Staubli VAL3: readText.dtx

public bool bBYPASS
public bool bCycle
public bool bCycleEnd
bool bGetSpeed = true
bool bMatlab
bool bReadEnd
bool bReadWait
public bool bResumeCycle
bool bTxtHeadOk
public bool bWriteEnd
frame fPrdFrame = {fatherId=world[0]}
jointRx jJointRead[100] = {j1=8.22, j2=20.1, j3=107.19, j4=-141.77, j5=44.38, j6=150.9}
public jointRx jPrdHome
mdesc mNomSpeed = {accel=16, vel=40, decel=16, tmax=80, blend=off, leave=20, reach=20}
public mdesc mSpdOfJnt[100]
  [0] = {accel=40, vel=40, decel=40, rmax=1000, tmax=40, blend=cartesian, leave=0, reach=2}
  [1] = {accel=30, vel=40, decel=30, rmax=1000, tmax=40, blend=cartesian, leave=0, reach=2}
  [2] = {accel=30, vel=40, decel=30, rmax=1000, tmax=15.702, blend=cartesian, leave=0, reach=2}
  [3] = {accel=30, vel=40, decel=30, rmax=1000, tmax=6.112, blend=cartesian, leave=0, reach=2}
  [4] = {accel=16, vel=40, decel=16, rmax=1000, tmax=200, blend=cartesian, leave=2, reach=2}
  [5] = {accel=16, vel=40, decel=16, rmax=1000, tmax=200, blend=cartesian, leave=2, reach=2}
  [6] = {accel=16, vel=40, decel=16, rmax=1000, tmax=200, blend=cartesian, leave=2, reach=2}
  [7] = {accel=16, vel=40, decel=16, rmax=1000, tmax=200, blend=cartesian, leave=2, reach=2}
  [8] = {accel=16, vel=40, decel=16, rmax=1000, tmax=200, blend=cartesian, leave=2, reach=2}
  [9] = {accel=16, vel=40, decel=16, rmax=1000, tmax=200, blend=cartesian, leave=2, reach=2}
  [10] = {accel=16, vel=40, decel=16, rmax=1000, tmax=200, blend=cartesian, leave=2, reach=2}
  [11] = {accel=16, vel=40, decel=16, rmax=1000, tmax=200, blend=cartesian, leave=2, reach=2}
  [12] = {accel=16, vel=40, decel=16, rmax=1000, tmax=200, blend=cartesian, leave=2, reach=2}
  [13] = {accel=16, vel=40, decel=16, rmax=1000, tmax=200, blend=cartesian, leave=2, reach=2}
  [14] = {accel=16, vel=40, decel=16, rmax=1000, tmax=200, blend=cartesian, leave=2, reach=2}
  [15] = {accel=16, vel=40, decel=16, rmax=1000, tmax=200, blend=cartesian, leave=2, reach=2}
  [16] = {accel=16, vel=40, decel=16, rmax=1000, tmax=200, blend=cartesian, leave=2, reach=2}
  [17] = {accel=16, vel=40, decel=16, rmax=1000, tmax=200, blend=cartesian, leave=2, reach=2}
  [18] = {accel=16, vel=40, decel=16, rmax=1000, tmax=200, blend=cartesian, leave=2, reach=2}
  [19] = {accel=16, vel=40, decel=16, rmax=1000, tmax=200, blend=cartesian, leave=2, reach=2}
  [20] = {accel=16, vel=40, decel=16, rmax=1000, tmax=200, blend=cartesian, leave=2, reach=2}
  [21] = {accel=16, vel=40, decel=16, rmax=1000, tmax=200, blend=cartesian, leave=2, reach=2}
  [22] = {accel=16, vel=40, decel=16, rmax=1000, tmax=200, blend=cartesian, leave=2, reach=2}
  [23] = {accel=16, vel=40, decel=16, rmax=1000, tmax=200, blend=cartesian, leave=2, reach=2}
  [24] = {accel=16, vel=40, decel=16, rmax=1000, tmax=200, blend=cartesian, leave=2, reach=2}
  [25] = {accel=16, vel=40, decel=16, rmax=1000, tmax=200, blend=cartesian, leave=2, reach=2}
  [26] = {accel=16, vel=40, decel=16, rmax=1000, tmax=200, blend=cartesian, leave=2, reach=2}
  [27] = {accel=16, vel=40, decel=16, rmax=1000, tmax=200, blend=cartesian, leave=2, reach=2}
  [28] = {accel=16, vel=40, decel=16, rmax=1000, tmax=200, blend=cartesian, leave=2, reach=2}
  [29] = {accel=16, vel=40, decel=16, rmax=1000, tmax=200, blend=cartesian, leave=2, reach=2}
  [30] = {accel=16, vel=40, decel=16, rmax=1000, tmax=200, blend=cartesian, leave=2, reach=2}
  [31] = {accel=16, vel=40, decel=16, rmax=1000, tmax=200, blend=cartesian, leave=2, reach=2}
  [32] = {accel=16, vel=40, decel=16, rmax=1000, tmax=200, blend=cartesian, leave=2, reach=2}
  [33] = {accel=16, vel=40, decel=16, rmax=1000, tmax=200, blend=cartesian, leave=2, reach=2}
  [34] = {accel=16, vel=40, decel=16, rmax=1000, tmax=200, blend=cartesian, leave=2, reach=2}
  [35] = {accel=16, vel=40, decel=16, rmax=1000, tmax=200, blend=cartesian, leave=2, reach=2}
  [36] = {accel=16, vel=40, decel=16, rmax=1000, tmax=200, blend=cartesian, leave=2, reach=2}
  [37] = {accel=16, vel=40, decel=16, rmax=1000, tmax=200, blend=cartesian, leave=2, reach=2}
  [38] = {accel=16, vel=40, decel=16, rmax=1000, tmax=200, blend=cartesian, leave=2, reach=2}
  [39] = {accel=16, vel=40, decel=16, rmax=1000, tmax=200, blend=cartesian, leave=2, reach=2}
  [40] = {accel=16, vel=40, decel=16, rmax=1000, tmax=200, blend=cartesian, leave=2, reach=2}
  [41] = {accel=16, vel=40, decel=16, rmax=1000, tmax=200, blend=cartesian, leave=2, reach=2}
  [42] = {accel=16, vel=40, decel=16, rmax=1000, tmax=200, blend=cartesian, leave=2, reach=2}
  [43] = {accel=16, vel=40, decel=16, rmax=1000, tmax=200, blend=cartesian, leave=2, reach=2}
  [44] = {accel=16, vel=40, decel=16, rmax=1000, tmax=200, blend=cartesian, leave=2, reach=2}
  [45] = {accel=16, vel=40, decel=16, rmax=1000, tmax=200, blend=cartesian, leave=2, reach=2}
  [46] = {accel=16, vel=40, decel=16, rmax=1000, tmax=200, blend=cartesian, leave=2, reach=2}
  [47] = {accel=16, vel=40, decel=16, rmax=1000, tmax=200, blend=cartesian, leave=2, reach=2}
  [48] = {accel=16, vel=40, decel=16, rmax=1000, tmax=200, blend=cartesian, leave=2, reach=2}
  [49] = {accel=16, vel=40, decel=16, rmax=1000, tmax=200, blend=cartesian, leave=2, reach=2}
  [50] = {accel=16, vel=40, decel=16, rmax=1000, tmax=200, blend=cartesian, leave=2, reach=2}
  [51] = {accel=16, vel=40, decel=16, rmax=1000, tmax=200, blend=cartesian, leave=2, reach=2}
  [52] = {accel=16, vel=40, decel=16, rmax=1000, tmax=200, blend=cartesian, leave=2, reach=2}
  [53] = {accel=16, vel=40, decel=16, rmax=1000, tmax=200, blend=cartesian, leave=2, reach=2}
  [54] = {accel=16, vel=40, decel=16, rmax=1000, tmax=200, blend=cartesian, leave=2, reach=2}
  [55] = {accel=16, vel=40, decel=16, rmax=1000, tmax=200, blend=cartesian, leave=2, reach=2}
  [56] = {accel=16, vel=40, decel=16, rmax=1000, tmax=200, blend=cartesian, leave=2, reach=2}
  [57] = {accel=16, vel=40, decel=16, rmax=1000, tmax=200, blend=cartesian, leave=2, reach=2}
  [58] = {accel=16, vel=40, decel=16, rmax=1000, tmax=200, blend=cartesian, leave=2, reach=2}
  [59] = {accel=16, vel=40, decel=16, rmax=1000, tmax=200, blend=cartesian, leave=2, reach=2}
  [60] = {accel=16, vel=40, decel=16, rmax=1000, tmax=200, blend=cartesian, leave=2, reach=2}
  [61] = {accel=16, vel=40, decel=16, rmax=1000, tmax=200, blend=cartesian, leave=2, reach=2}
  [62] = {accel=16, vel=40, decel=16, rmax=1000, tmax=200, blend=cartesian, leave=2, reach=2}
  [63] = {accel=16, vel=40, decel=16, rmax=1000, tmax=200, blend=cartesian, leave=2, reach=2}
  [64] = {accel=16, vel=40, decel=16, rmax=1000, tmax=200, blend=cartesian, leave=2, reach=2}
  [65] = {accel=16, vel=40, decel=16, rmax=1000, tmax=200, blend=cartesian, leave=2, reach=2}
  [66] = {accel=16, vel=40, decel=16, rmax=1000, tmax=200, blend=cartesian, leave=2, reach=2}
  [67] = {accel=16, vel=40, decel=16, rmax=1000, tmax=200, blend=cartesian, leave=2, reach=2}
  [68] = {accel=16, vel=40, decel=16, rmax=1000, tmax=200, blend=cartesian, leave=2, reach=2}
  [69] = {accel=16, vel=40, decel=16, rmax=1000, tmax=200, blend=cartesian, leave=2, reach=2}
  [70] = {accel=16, vel=40, decel=16, rmax=1000, tmax=200, blend=cartesian, leave=2, reach=2}
  [71] = {accel=16, vel=40, decel=16, rmax=1000, tmax=200, blend=cartesian, leave=2, reach=2}
  [72] = {accel=16, vel=40, decel=16, rmax=1000, tmax=200, blend=cartesian, leave=2, reach=2}
  [73] = {accel=16, vel=40, decel=16, rmax=1000, tmax=200, blend=cartesian, leave=2, reach=2}
  [74] = {accel=16, vel=40, decel=16, rmax=1000, tmax=200, blend=cartesian, leave=2, reach=2}
  [75] = {accel=16, vel=40, decel=16, rmax=1000, tmax=200, blend=cartesian, leave=2, reach=2}
  [76] = {accel=16, vel=40, decel=16, rmax=1000, tmax=200, blend=cartesian, leave=2, reach=2}
  [77] = {accel=16, vel=40, decel=16, rmax=1000, tmax=200, blend=cartesian, leave=2, reach=2}
  [78] = {accel=16, vel=40, decel=16, rmax=1000, tmax=200, blend=cartesian, leave=2, reach=2}
  [79] = {accel=16, vel=40, decel=16, rmax=1000, tmax=200, blend=cartesian, leave=2, reach=2}
  [80] = {accel=16, vel=40, decel=16, rmax=1000, tmax=200, blend=cartesian, leave=2, reach=2}
  [81] = {accel=16, vel=40, decel=16, rmax=1000, tmax=200, blend=cartesian, leave=2, reach=2}
  [82] = {accel=16, vel=40, decel=16, rmax=1000, tmax=200, blend=cartesian, leave=2, reach=2}
  [83] = {accel=16, vel=40, decel=16, rmax=1000, tmax=200, blend=cartesian, leave=2, reach=2}
  [84] = {accel=16, vel=40, decel=16, rmax=1000, tmax=200, blend=cartesian, leave=2, reach=2}
  [85] = {accel=16, vel=40, decel=16, rmax=1000, tmax=200, blend=cartesian, leave=2, reach=2}
  [86] = {accel=16, vel=40, decel=16, rmax=1000, tmax=200, blend=cartesian, leave=2, reach=2}
  [87] = {accel=16, vel=40, decel=16, rmax=1000, tmax=200, blend=cartesian, leave=2, reach=2}
  [88] = {accel=16, vel=40, decel=16, rmax=1000, tmax=200, blend=cartesian, leave=2, reach=2}
  [89] = {accel=16, vel=40, decel=16, rmax=1000, tmax=200, blend=cartesian, leave=2, reach=2}
  [90] = {accel=16, vel=40, decel=16, rmax=1000, tmax=200, blend=cartesian, leave=2, reach=2}
  [91] = {accel=16, vel=40, decel=16, rmax=1000, tmax=200, blend=cartesian, leave=2, reach=2}
  [92] = {accel=16, vel=40, decel=16, rmax=1000, tmax=200, blend=cartesian, leave=2, reach=2}
  [93] = {accel=16, vel=40, decel=16, rmax=1000, tmax=200, blend=cartesian, leave=2, reach=2}
  [94] = {accel=16, vel=40, decel=16, rmax=1000, tmax=200, blend=cartesian, leave=2, reach=2}
  [95] = {accel=16, vel=40, decel=16, rmax=1000, tmax=200, blend=cartesian, leave=2, reach=2}
  [96] = {accel=16, vel=40, decel=16, rmax=1000, tmax=200, blend=cartesian, leave=2, reach=2}
  [97] = {accel=16, vel=40, decel=16, rmax=1000, tmax=200, blend=cartesian, leave=2, reach=2}
  [98] = {accel=16, vel=40, decel=16, rmax=1000, tmax=200, blend=cartesian, leave=2, reach=2}
  [99] = {accel=16, vel=40, decel=16, rmax=1000, tmax=200, blend=cartesian, leave=2, reach=2}
public mdesc mSpdOfPt[1000]
  [0] = {accel=30, decel=30, tmax=100, leave=0, reach=0.5}
  [1] = {accel=80, decel=80, tmax=40, leave=0.5, reach=0.5}
  [2] = {accel=80, decel=80, tmax=20, leave=2, reach=0.5}
  [3] = {accel=80, decel=80, tmax=6.283, leave=0, reach=0.5}
  [4] = {accel=80, decel=80, tmax=9.415, leave=0, reach=0.5}
  [5] = {accel=80, decel=80, tmax=9.426, leave=0, reach=0.5}
  [6] = {accel=80, decel=80, tmax=9.491, leave=0, reach=0.5}
  [7] = {accel=80, decel=80, tmax=9.63, leave=0, reach=0.5}
  [8] = {accel=80, decel=80, tmax=9.837, leave=0, reach=0.5}
  [9] = {accel=80, decel=80, tmax=10.085, leave=0, reach=0.5}
  [10] = {accel=80, decel=80, tmax=10.343, leave=0, reach=0.5}
  [11] = {accel=80, decel=80, tmax=10.597, leave=0, reach=0.5}
  [12] = {accel=80, decel=80, tmax=10.851, leave=0, reach=0.5}
  [13] = {accel=80, decel=80, tmax=11.121, leave=0, reach=0.5}
  [14] = {accel=80, decel=80, tmax=11.43, leave=0, reach=0.5}
  [15] = {accel=80, decel=80, tmax=11.774, leave=0, reach=0.5}
  [16] = {accel=80, decel=80, tmax=12.135, leave=0, reach=0.5}
  [17] = {accel=80, decel=80, tmax=12.558, leave=0, reach=0.5}
  [18] = {accel=80, decel=80, tmax=13.049, leave=0, reach=0.5}
  [19] = {accel=80, decel=80, tmax=13.543, leave=0, reach=0.5}
  [20] = {accel=80, decel=80, tmax=14.016, leave=0, reach=0.5}
  [21] = {accel=80, decel=80, tmax=14.458, leave=0, reach=0.5}
  [22] = {accel=80, decel=80, tmax=14.885, leave=0, reach=0.5}
  [23] = {accel=80, decel=80, tmax=15.328, leave=0, reach=0.5}
  [24] = {accel=80, decel=80, tmax=15.823, leave=0, reach=0.5}
  [25] = {accel=80, decel=80, tmax=16.391, leave=0, reach=0.5}
  [26] = {accel=80, decel=80, tmax=17.025, leave=0, reach=0.5}
  [27] = {accel=80, decel=80, tmax=17.694, leave=0, reach=0.5}
  [28] = {accel=80, decel=80, tmax=80, leave=0, reach=0.5}
  [29] = {accel=80, decel=80, tmax=22.598, leave=0, reach=0.5}
  [30] = {accel=80, decel=80, tmax=22.402, leave=0, reach=0.5}
  [31] = {accel=80, decel=80, tmax=21.992, leave=0, reach=0.5}
  [32] = {accel=80, decel=80, tmax=21.406, leave=0, reach=0.5}
  [33] = {accel=80, decel=80, tmax=20.689, leave=0, reach=0.5}
  [34] = {accel=80, decel=80, tmax=19.887, leave=0, reach=0.5}
  [35] = {accel=80, decel=80, tmax=19.047, leave=0, reach=0.5}
  [36] = {accel=80, decel=80, tmax=18.222, leave=0, reach=0.5}
  [37] = {accel=80, decel=80, tmax=17.459, leave=0, reach=0.5}
  [38] = {accel=80, decel=80, tmax=16.784, leave=0, reach=0.5}
  [39] = {accel=80, decel=80, tmax=16.194, leave=0, reach=0.5}
  [40] = {accel=80, decel=80, tmax=15.663, leave=0, reach=0.5}
  [41] = {accel=80, decel=80, tmax=15.153, leave=0, reach=0.5}
  [42] = {accel=80, decel=80, tmax=14.634, leave=0, reach=0.5}
  [43] = {accel=80, decel=80, tmax=14.096, leave=0, reach=0.5}
  [44] = {accel=80, decel=80, tmax=13.551, leave=0, reach=0.5}
  [45] = {accel=80, decel=80, tmax=13.023, leave=0, reach=0.5}
  [46] = {accel=80, decel=80, tmax=12.575, leave=0, reach=0.5}
  [47] = {accel=80, decel=80, tmax=12.194, leave=0, reach=0.5}
  [48] = {accel=80, decel=80, tmax=11.83, leave=0, reach=0.5}
  [49] = {accel=80, decel=80, tmax=11.503, leave=0, reach=0.5}
  [50] = {accel=80, decel=80, tmax=11.215, leave=0, reach=0.5}
  [51] = {accel=80, decel=80, tmax=10.948, leave=0, reach=0.5}
  [52] = {accel=80, decel=80, tmax=10.683, leave=0, reach=0.5}
  [53] = {accel=80, decel=80, tmax=10.416, leave=0, reach=0.5}
  [54] = {accel=80, decel=80, tmax=10.16, leave=0, reach=0.5}
  [55] = {accel=80, decel=80, tmax=9.943, leave=0, reach=0.5}
  [56] = {accel=80, decel=80, tmax=9.794, leave=0, reach=0.5}
  [57] = {accel=80, decel=80, tmax=9.721, leave=0, reach=0.5}
  [58] = {accel=80, decel=80, tmax=9.707, leave=0, reach=0.5}
  [59] = {accel=80, decel=80, tmax=9.72, leave=0, reach=0.5}
  [60] = {accel=80, decel=80, tmax=9.72, leave=0, reach=0.5}
  [61] = {accel=80, decel=80, tmax=9.688, leave=0, reach=0.5}
  [62] = {accel=80, decel=80, tmax=9.617, leave=0, reach=0.5}
  [63] = {accel=80, decel=80, tmax=9.515, leave=0, reach=0.5}
  [64] = {accel=80, decel=80, tmax=9.389, leave=0, reach=0.5}
  [65] = {accel=80, decel=80, tmax=46.527, leave=0, reach=0.5}
  [66] = {accel=80, decel=80, tmax=8.998, leave=0, reach=0.5}
  [67] = {accel=80, decel=80, tmax=9.118, leave=0, reach=0.5}
  [68] = {accel=80, decel=80, tmax=9.246, leave=0, reach=0.5}
  [69] = {accel=80, decel=80, tmax=9.386, leave=0, reach=0.5}
  [70] = {accel=80, decel=80, tmax=9.534, leave=0, reach=0.5}
  [71] = {accel=80, decel=80, tmax=9.678, leave=0, reach=0.5}
  [72] = {accel=80, decel=80, tmax=9.805, leave=0, reach=0.5}
  [73] = {accel=80, decel=80, tmax=9.903, leave=0, reach=0.5}
  [74] = {accel=80, decel=80, tmax=9.967, leave=0, reach=0.5}
  [75] = {accel=80, decel=80, tmax=9.994, leave=0, reach=0.5}
  [76] = {accel=80, decel=80, tmax=9.995, leave=0, reach=0.5}
  [77] = {accel=80, decel=80, tmax=9.992, leave=0, reach=0.5}
  [78] = {accel=80, decel=80, tmax=10.02, leave=0, reach=0.5}
  [79] = {accel=80, decel=80, tmax=10.106, leave=0, reach=0.5}
  [80] = {accel=80, decel=80, tmax=10.26, leave=0, reach=0.5}
  [81] = {accel=80, decel=80, tmax=10.472, leave=0, reach=0.5}
  [82] = {accel=80, decel=80, tmax=10.718, leave=0, reach=0.5}
  [83] = {accel=80, decel=80, tmax=10.977, leave=0, reach=0.5}
  [84] = {accel=80, decel=80, tmax=11.242, leave=0, reach=0.5}
  [85] = {accel=80, decel=80, tmax=11.521, leave=0, reach=0.5}
  [86] = {accel=80, decel=80, tmax=11.83, leave=0, reach=0.5}
  [87] = {accel=80, decel=80, tmax=12.182, leave=0, reach=0.5}
  [88] = {accel=80, decel=80, tmax=12.568, leave=0, reach=0.5}
  [89] = {accel=80, decel=80, tmax=12.965, leave=0, reach=0.5}
  [90] = {accel=80, decel=80, tmax=13.429, leave=0, reach=0.5}
  [91] = {accel=80, decel=80, tmax=13.979, leave=0, reach=0.5}
  [92] = {accel=80, decel=80, tmax=14.561, leave=0, reach=0.5}
  [93] = {accel=80, decel=80, tmax=15.156, leave=0, reach=0.5}
  [94] = {accel=80, decel=80, tmax=15.752, leave=0, reach=0.5}
  [95] = {accel=80, decel=80, tmax=16.352, leave=0, reach=0.5}
  [96] = {accel=80, decel=80, tmax=16.979, leave=0, reach=0.5}
  [97] = {accel=80, decel=80, tmax=17.664, leave=0, reach=0.5}
  [98] = {accel=80, decel=80, tmax=18.437, leave=0, reach=0.5}
  [99] = {accel=80, decel=80, tmax=19.31, leave=0, reach=0.5}
  [100] = {accel=80, decel=80, tmax=20.273, leave=0, reach=0.5}
  [101] = {accel=80, decel=80, tmax=21.286, leave=0, reach=0.5}
  [102] = {accel=80, decel=80, tmax=22.298, leave=0, reach=0.5}
  [103] = {accel=80, decel=80, tmax=23.255, leave=0, reach=0.5}
  [104] = {accel=80, decel=80, tmax=24.103, leave=0, reach=0.5}
  [105] = {accel=80, decel=80, tmax=24.781, leave=0, reach=0.5}
  [106] = {accel=80, decel=80, tmax=25.228, leave=0, reach=0.5}
  [107] = {accel=80, decel=80, tmax=25.404, leave=0, reach=0.5}
  [108] = {accel=80, decel=80, tmax=25.299, leave=0, reach=0.5}
  [109] = {accel=80, decel=80, tmax=24.922, leave=0, reach=0.5}
  [110] = {accel=80, decel=80, tmax=24.286, leave=0, reach=0.5}
  [111] = {accel=80, decel=80, tmax=75.027, leave=0, reach=0.5}
  [112] = {accel=80, decel=80, tmax=24.232, leave=0, reach=0.5}
  [113] = {accel=80, decel=80, tmax=25.564, leave=0, reach=0.5}
  [114] = {accel=80, decel=80, tmax=26.713, leave=0, reach=0.5}
  [115] = {accel=80, decel=80, tmax=27.589, leave=0, reach=0.5}
  [116] = {accel=80, decel=80, tmax=28.14, leave=0, reach=0.5}
  [117] = {accel=80, decel=80, tmax=28.354, leave=0, reach=0.5}
  [118] = {accel=80, decel=80, tmax=28.23, leave=0, reach=0.5}
  [119] = {accel=80, decel=80, tmax=27.776, leave=0, reach=0.5}
  [120] = {accel=80, decel=80, tmax=27.029, leave=0, reach=0.5}
  [121] = {accel=80, decel=80, tmax=26.056, leave=0, reach=0.5}
  [122] = {accel=80, decel=80, tmax=24.937, leave=0, reach=0.5}
  [123] = {accel=80, decel=80, tmax=23.743, leave=0, reach=0.5}
  [124] = {accel=80, decel=80, tmax=22.534, leave=0, reach=0.5}
  [125] = {accel=80, decel=80, tmax=21.368, leave=0, reach=0.5}
  [126] = {accel=80, decel=80, tmax=20.288, leave=0, reach=0.5}
  [127] = {accel=80, decel=80, tmax=19.318, leave=0, reach=0.5}
  [128] = {accel=80, decel=80, tmax=18.454, leave=0, reach=0.5}
  [129] = {accel=80, decel=80, tmax=17.673, leave=0, reach=0.5}
  [130] = {accel=80, decel=80, tmax=16.951, leave=0, reach=0.5}
  [131] = {accel=80, decel=80, tmax=16.265, leave=0, reach=0.5}
  [132] = {accel=80, decel=80, tmax=15.601, leave=0, reach=0.5}
  [133] = {accel=80, decel=80, tmax=14.96, leave=0, reach=0.5}
  [134] = {accel=80, decel=80, tmax=14.352, leave=0, reach=0.5}
  [135] = {accel=80, decel=80, tmax=13.787, leave=0, reach=0.5}
  [136] = {accel=80, decel=80, tmax=13.313, leave=0, reach=0.5}
  [137] = {accel=80, decel=80, tmax=12.9, leave=0, reach=0.5}
  [138] = {accel=80, decel=80, tmax=12.491, leave=0, reach=0.5}
  [139] = {accel=80, decel=80, tmax=12.111, leave=0, reach=0.5}
  [140] = {accel=80, decel=80, tmax=11.779, leave=0, reach=0.5}
  [141] = {accel=80, decel=80, tmax=11.485, leave=0, reach=0.5}
  [142] = {accel=80, decel=80, tmax=11.218, leave=0, reach=0.5}
  [143] = {accel=80, decel=80, tmax=10.971, leave=0, reach=0.5}
  [144] = {accel=80, decel=80, tmax=10.743, leave=0, reach=0.5}
  [145] = {accel=80, decel=80, tmax=10.546, leave=0, reach=0.5}
  [146] = {accel=80, decel=80, tmax=10.395, leave=0, reach=0.5}
  [147] = {accel=80, decel=80, tmax=10.3, leave=0, reach=0.5}
  [148] = {accel=80, decel=80, tmax=10.256, leave=0, reach=0.5}
  [149] = {accel=80, decel=80, tmax=10.244, leave=0, reach=0.5}
  [150] = {accel=80, decel=80, tmax=10.237, leave=0, reach=0.5}
  [151] = {accel=80, decel=80, tmax=10.212, leave=0, reach=0.5}
  [152] = {accel=80, decel=80, tmax=10.153, leave=0, reach=0.5}
  [153] = {accel=80, decel=80, tmax=10.056, leave=0, reach=0.5}
  [154] = {accel=80, decel=80, tmax=9.924, leave=0, reach=0.5}
  [155] = {accel=80, decel=80, tmax=9.77, leave=0, reach=0.5}
  [156] = {accel=80, decel=80, tmax=9.616, leave=0, reach=0.5}
  [157] = {accel=80, decel=80, tmax=9.484, leave=0, reach=0.5}
  [158] = {accel=80, decel=80, tmax=9.383, leave=0, reach=0.5}
  [159] = {accel=80, decel=80, tmax=9.304, leave=0, reach=0.5}
  [160] = {accel=80, decel=80, tmax=9.229, leave=0, reach=0.5}
  [161] = {accel=80, decel=80, tmax=9.137, leave=0, reach=0.5}
  [162] = {accel=80, decel=80, tmax=9.012, leave=0, reach=0.5}
  [163] = {accel=80, decel=80, tmax=28.213, leave=0, reach=0.5}
  [164] = {accel=80, decel=80, tmax=8.988, leave=0, reach=0.5}
  [165] = {accel=80, decel=80, tmax=9.149, leave=0, reach=0.5}
  [166] = {accel=80, decel=80, tmax=9.308, leave=0, reach=0.5}
  [167] = {accel=80, decel=80, tmax=9.436, leave=0, reach=0.5}
  [168] = {accel=80, decel=80, tmax=9.518, leave=0, reach=0.5}
  [169] = {accel=80, decel=80, tmax=9.559, leave=0, reach=0.5}
  [170] = {accel=80, decel=80, tmax=9.58, leave=0, reach=0.5}
  [171] = {accel=80, decel=80, tmax=9.614, leave=0, reach=0.5}
  [172] = {accel=80, decel=80, tmax=9.691, leave=0, reach=0.5}
  [173] = {accel=80, decel=80, tmax=9.819, leave=0, reach=0.5}
  [174] = {accel=80, decel=80, tmax=9.982, leave=0, reach=0.5}
  [175] = {accel=80, decel=80, tmax=10.147, leave=0, reach=0.5}
  [176] = {accel=80, decel=80, tmax=10.285, leave=0, reach=0.5}
  [177] = {accel=80, decel=80, tmax=10.38, leave=0, reach=0.5}
  [178] = {accel=80, decel=80, tmax=10.433, leave=0, reach=0.5}
  [179] = {accel=80, decel=80, tmax=10.454, leave=0, reach=0.5}
  [180] = {accel=80, decel=80, tmax=10.462, leave=0, reach=0.5}
  [181] = {accel=80, decel=80, tmax=10.479, leave=0, reach=0.5}
  [182] = {accel=80, decel=80, tmax=10.528, leave=0, reach=0.5}
  [183] = {accel=80, decel=80, tmax=10.621, leave=0, reach=0.5}
  [184] = {accel=80, decel=80, tmax=10.76, leave=0, reach=0.5}
  [185] = {accel=80, decel=80, tmax=10.941, leave=0, reach=0.5}
  [186] = {accel=80, decel=80, tmax=11.155, leave=0, reach=0.5}
  [187] = {accel=80, decel=80, tmax=11.399, leave=0, reach=0.5}
  [188] = {accel=80, decel=80, tmax=11.674, leave=0, reach=0.5}
  [189] = {accel=80, decel=80, tmax=11.989, leave=0, reach=0.5}
  [190] = {accel=80, decel=80, tmax=12.349, leave=0, reach=0.5}
  [191] = {accel=80, decel=80, tmax=12.758, leave=0, reach=0.5}
  [192] = {accel=80, decel=80, tmax=13.191, leave=0, reach=0.5}
  [193] = {accel=80, decel=80, tmax=13.618, leave=0, reach=0.5}
  [194] = {accel=80, decel=80, tmax=14.103, leave=0, reach=0.5}
  [195] = {accel=80, decel=80, tmax=14.68, leave=0, reach=0.5}
  [196] = {accel=80, decel=80, tmax=15.307, leave=0, reach=0.5}
  [197] = {accel=80, decel=80, tmax=15.981, leave=0, reach=0.5}
  [198] = {accel=80, decel=80, tmax=16.697, leave=0, reach=0.5}
  [199] = {accel=80, decel=80, tmax=17.456, leave=0, reach=0.5}
  [200] = {accel=80, decel=80, tmax=18.265, leave=0, reach=0.5}
  [201] = {accel=80, decel=80, tmax=19.14, leave=0, reach=0.5}
  [202] = {accel=80, decel=80, tmax=20.1, leave=0, reach=0.5}
  [203] = {accel=80, decel=80, tmax=21.165, leave=0, reach=0.5}
  [204] = {accel=80, decel=80, tmax=22.354, leave=0, reach=0.5}
  [205] = {accel=80, decel=80, tmax=23.661, leave=0, reach=0.5}
  [206] = {accel=80, decel=80, tmax=25.052, leave=0, reach=0.5}
  [207] = {accel=80, decel=80, tmax=26.473, leave=0, reach=0.5}
  [208] = {accel=80, decel=80, tmax=27.858, leave=0, reach=0.5}
  [209] = {accel=80, decel=80, tmax=29.13, leave=0, reach=0.5}
  [210] = {accel=80, decel=80, tmax=30.198, leave=0, reach=0.5}
  [211] = {accel=80, decel=80, tmax=30.973, leave=0, reach=0.5}
  [212] = {accel=80, decel=80, tmax=31.392, leave=0, reach=0.5}
  [213] = {accel=80, decel=80, tmax=31.427, leave=0, reach=0.5}
  [214] = {accel=80, decel=80, tmax=31.052, leave=0, reach=0.5}
  [215] = {accel=80, decel=80, tmax=30.253, leave=0, reach=0.5}
  [216] = {accel=80, decel=80, tmax=29.062, leave=0, reach=0.5}
  [217] = {accel=80, decel=80, tmax=27.585, leave=0, reach=0.5}
  [218] = {accel=80, decel=80, tmax=25.953, leave=0, reach=0.5}
  [219] = {accel=80, decel=80, tmax=24.265, leave=0, reach=0.5}
  [220] = {accel=80, decel=80, tmax=22.574, leave=0, reach=0.5}
  [221] = {accel=80, decel=80, tmax=63.913, leave=0, reach=0.5}
  [222] = {accel=80, decel=80, tmax=19.723, leave=0, reach=0.5}
  [223] = {accel=80, decel=80, tmax=21.535, leave=0, reach=0.5}
  [224] = {accel=80, decel=80, tmax=23.435, leave=0, reach=0.5}
  [225] = {accel=80, decel=80, tmax=25.393, leave=0, reach=0.5}
  [226] = {accel=80, decel=80, tmax=27.381, leave=0, reach=0.5}
  [227] = {accel=80, decel=80, tmax=29.346, leave=0, reach=0.5}
  [228] = {accel=80, decel=80, tmax=31.196, leave=0, reach=0.5}
  [229] = {accel=80, decel=80, tmax=32.785, leave=0, reach=0.5}
  [230] = {accel=80, decel=80, tmax=33.949, leave=0, reach=0.5}
  [231] = {accel=80, decel=80, tmax=34.591, leave=0, reach=0.5}
  [232] = {accel=80, decel=80, tmax=34.718, leave=0, reach=0.5}
  [233] = {accel=80, decel=80, tmax=34.385, leave=0, reach=0.5}
  [234] = {accel=80, decel=80, tmax=33.637, leave=0, reach=0.5}
  [235] = {accel=80, decel=80, tmax=32.521, leave=0, reach=0.5}
  [236] = {accel=80, decel=80, tmax=31.12, leave=0, reach=0.5}
  [237] = {accel=80, decel=80, tmax=29.544, leave=0, reach=0.5}
  [238] = {accel=80, decel=80, tmax=27.893, leave=0, reach=0.5}
  [239] = {accel=80, decel=80, tmax=26.25, leave=0, reach=0.5}
  [240] = {accel=80, decel=80, tmax=24.68, leave=0, reach=0.5}
  [241] = {accel=80, decel=80, tmax=23.233, leave=0, reach=0.5}
  [242] = {accel=80, decel=80, tmax=21.927, leave=0, reach=0.5}
  [243] = {accel=80, decel=80, tmax=20.755, leave=0, reach=0.5}
  [244] = {accel=80, decel=80, tmax=19.695, leave=0, reach=0.5}
  [245] = {accel=80, decel=80, tmax=18.727, leave=0, reach=0.5}
  [246] = {accel=80, decel=80, tmax=17.841, leave=0, reach=0.5}
  [247] = {accel=80, decel=80, tmax=17.027, leave=0, reach=0.5}
  [248] = {accel=80, decel=80, tmax=16.274, leave=0, reach=0.5}
  [249] = {accel=80, decel=80, tmax=15.579, leave=0, reach=0.5}
  [250] = {accel=80, decel=80, tmax=14.94, leave=0, reach=0.5}
  [251] = {accel=80, decel=80, tmax=14.354, leave=0, reach=0.5}
  [252] = {accel=80, decel=80, tmax=13.859, leave=0, reach=0.5}
  [253] = {accel=80, decel=80, tmax=13.416, leave=0, reach=0.5}
  [254] = {accel=80, decel=80, tmax=12.961, leave=0, reach=0.5}
  [255] = {accel=80, decel=80, tmax=12.525, leave=0, reach=0.5}
  [256] = {accel=80, decel=80, tmax=12.137, leave=0, reach=0.5}
  [257] = {accel=80, decel=80, tmax=11.798, leave=0, reach=0.5}
  [258] = {accel=80, decel=80, tmax=11.507, leave=0, reach=0.5}
  [259] = {accel=80, decel=80, tmax=11.259, leave=0, reach=0.5}
  [260] = {accel=80, decel=80, tmax=11.051, leave=0, reach=0.5}
  [261] = {accel=80, decel=80, tmax=10.884, leave=0, reach=0.5}
  [262] = {accel=80, decel=80, tmax=10.761, leave=0, reach=0.5}
  [263] = {accel=80, decel=80, tmax=10.683, leave=0, reach=0.5}
  [264] = {accel=80, decel=80, tmax=10.647, leave=0, reach=0.5}
  [265] = {accel=80, decel=80, tmax=10.64, leave=0, reach=0.5}
  [266] = {accel=80, decel=80, tmax=10.643, leave=0, reach=0.5}
  [267] = {accel=80, decel=80, tmax=10.634, leave=0, reach=0.5}
  [268] = {accel=80, decel=80, tmax=10.593, leave=0, reach=0.5}
  [269] = {accel=80, decel=80, tmax=10.507, leave=0, reach=0.5}
  [270] = {accel=80, decel=80, tmax=10.374, leave=0, reach=0.5}
  [271] = {accel=80, decel=80, tmax=10.205, leave=0, reach=0.5}
  [272] = {accel=80, decel=80, tmax=10.035, leave=0, reach=0.5}
  [273] = {accel=80, decel=80, tmax=9.904, leave=0, reach=0.5}
  [274] = {accel=80, decel=80, tmax=9.84, leave=0, reach=0.5}
  [275] = {accel=80, decel=80, tmax=9.839, leave=0, reach=0.5}
  [276] = {accel=80, decel=80, tmax=9.866, leave=0, reach=0.5}
  [277] = {accel=80, decel=80, tmax=9.877, leave=0, reach=0.5}
  [278] = {accel=80, decel=80, tmax=9.841, leave=0, reach=0.5}
  [279] = {accel=80, decel=80, tmax=9.75, leave=0, reach=0.5}
  [280] = {accel=80, decel=80, tmax=9.622, leave=0, reach=0.5}
  [281] = {accel=80, decel=80, tmax=9.483, leave=0, reach=0.5}
  [282] = {accel=80, decel=80, tmax=9.36, leave=0, reach=0.5}
  [283] = {accel=80, decel=80, tmax=9.27, leave=0, reach=0.5}
  [284] = {accel=80, decel=80, tmax=9.213, leave=0, reach=0.5}
  [285] = {accel=80, decel=80, tmax=21.042, leave=0, reach=0.5}
  [286] = {accel=80, decel=80, tmax=9.663, leave=0, reach=0.5}
  [287] = {accel=80, decel=80, tmax=9.685, leave=0, reach=0.5}
  [288] = {accel=80, decel=80, tmax=9.712, leave=0, reach=0.5}
  [289] = {accel=80, decel=80, tmax=9.76, leave=0, reach=0.5}
  [290] = {accel=80, decel=80, tmax=9.837, leave=0, reach=0.5}
  [291] = {accel=80, decel=80, tmax=9.942, leave=0, reach=0.5}
  [292] = {accel=80, decel=80, tmax=10.057, leave=0, reach=0.5}
  [293] = {accel=80, decel=80, tmax=10.157, leave=0, reach=0.5}
  [294] = {accel=80, decel=80, tmax=10.214, leave=0, reach=0.5}
  [295] = {accel=80, decel=80, tmax=10.212, leave=0, reach=0.5}
  [296] = {accel=80, decel=80, tmax=10.163, leave=0, reach=0.5}
  [297] = {accel=80, decel=80, tmax=10.107, leave=0, reach=0.5}
  [298] = {accel=80, decel=80, tmax=10.096, leave=0, reach=0.5}
  [299] = {accel=80, decel=80, tmax=10.159, leave=0, reach=0.5}
  [300] = {accel=80, decel=80, tmax=10.292, leave=0, reach=0.5}
  [301] = {accel=80, decel=80, tmax=10.456, leave=0, reach=0.5}
  [302] = {accel=80, decel=80, tmax=10.607, leave=0, reach=0.5}
  [303] = {accel=80, decel=80, tmax=10.718, leave=0, reach=0.5}
  [304] = {accel=80, decel=80, tmax=10.78, leave=0, reach=0.5}
  [305] = {accel=80, decel=80, tmax=10.8, leave=0, reach=0.5}
  [306] = {accel=80, decel=80, tmax=10.789, leave=0, reach=0.5}
  [307] = {accel=80, decel=80, tmax=10.764, leave=0, reach=0.5}
  [308] = {accel=80, decel=80, tmax=10.748, leave=0, reach=0.5}
  [309] = {accel=80, decel=80, tmax=10.761, leave=0, reach=0.5}
  [310] = {accel=80, decel=80, tmax=10.815, leave=0, reach=0.5}
  [311] = {accel=80, decel=80, tmax=10.918, leave=0, reach=0.5}
  [312] = {accel=80, decel=80, tmax=11.071, leave=0, reach=0.5}
  [313] = {accel=80, decel=80, tmax=11.275, leave=0, reach=0.5}
  [314] = {accel=80, decel=80, tmax=11.531, leave=0, reach=0.5}
  [315] = {accel=80, decel=80, tmax=11.838, leave=0, reach=0.5}
  [316] = {accel=80, decel=80, tmax=12.198, leave=0, reach=0.5}
  [317] = {accel=80, decel=80, tmax=12.61, leave=0, reach=0.5}
  [318] = {accel=80, decel=80, tmax=13.068, leave=0, reach=0.5}
  [319] = {accel=80, decel=80, tmax=13.541, leave=0, reach=0.5}
  [320] = {accel=80, decel=80, tmax=13.996, leave=0, reach=0.5}
  [321] = {accel=80, decel=80, tmax=14.5, leave=0, reach=0.5}
  [322] = {accel=80, decel=80, tmax=15.093, leave=0, reach=0.5}
  [323] = {accel=80, decel=80, tmax=15.736, leave=0, reach=0.5}
  [324] = {accel=80, decel=80, tmax=16.439, leave=0, reach=0.5}
  [325] = {accel=80, decel=80, tmax=17.212, leave=0, reach=0.5}
  [326] = {accel=80, decel=80, tmax=18.066, leave=0, reach=0.5}
  [327] = {accel=80, decel=80, tmax=19.014, leave=0, reach=0.5}
  [328] = {accel=80, decel=80, tmax=20.065, leave=0, reach=0.5}
  [329] = {accel=80, decel=80, tmax=21.228, leave=0, reach=0.5}
  [330] = {accel=80, decel=80, tmax=22.515, leave=0, reach=0.5}
  [331] = {accel=80, decel=80, tmax=23.948, leave=0, reach=0.5}
  [332] = {accel=80, decel=80, tmax=25.544, leave=0, reach=0.5}
  [333] = {accel=80, decel=80, tmax=27.295, leave=0, reach=0.5}
  [334] = {accel=80, decel=80, tmax=29.164, leave=0, reach=0.5}
  [335] = {accel=80, decel=80, tmax=31.092, leave=0, reach=0.5}
  [336] = {accel=80, decel=80, tmax=32.994, leave=0, reach=0.5}
  [337] = {accel=80, decel=80, tmax=34.75, leave=0, reach=0.5}
  [338] = {accel=80, decel=80, tmax=36.227, leave=0, reach=0.5}
  [339] = {accel=80, decel=80, tmax=37.319, leave=0, reach=0.5}
  [340] = {accel=80, decel=80, tmax=37.967, leave=0, reach=0.5}
  [341] = {accel=80, decel=80, tmax=38.114, leave=0, reach=0.5}
  [342] = {accel=80, decel=80, tmax=37.673, leave=0, reach=0.5}
  [343] = {accel=80, decel=80, tmax=36.585, leave=0, reach=0.5}
  [344] = {accel=80, decel=80, tmax=34.912, leave=0, reach=0.5}
  [345] = {accel=80, decel=80, tmax=32.836, leave=0, reach=0.5}
  [346] = {accel=80, decel=80, tmax=30.562, leave=0, reach=0.5}
  [347] = {accel=80, decel=80, tmax=28.246, leave=0, reach=0.5}
  [348] = {accel=80, decel=80, tmax=25.983, leave=0, reach=0.5}
  [349] = {accel=80, decel=80, tmax=23.824, leave=0, reach=0.5}
  [350] = {accel=80, decel=80, tmax=21.799, leave=0, reach=0.5}
  [351] = {accel=80, decel=80, tmax=19.926, leave=0, reach=0.5}
  [352] = {accel=80, decel=80, tmax=18.221, leave=0, reach=0.5}
  [353] = {accel=80, decel=80, tmax=50.879, leave=0, reach=0.5}
  [354] = {accel=80, decel=80, tmax=15.54, leave=0, reach=0.5}
  [355] = {accel=80, decel=80, tmax=16.856, leave=0, reach=0.5}
  [356] = {accel=80, decel=80, tmax=18.338, leave=0, reach=0.5}
  [357] = {accel=80, decel=80, tmax=19.996, leave=0, reach=0.5}
  [358] = {accel=80, decel=80, tmax=21.835, leave=0, reach=0.5}
  [359] = {accel=80, decel=80, tmax=23.857, leave=0, reach=0.5}
  [360] = {accel=80, decel=80, tmax=26.061, leave=0, reach=0.5}
  [361] = {accel=80, decel=80, tmax=28.443, leave=0, reach=0.5}
  [362] = {accel=80, decel=80, tmax=30.983, leave=0, reach=0.5}
  [363] = {accel=80, decel=80, tmax=33.616, leave=0, reach=0.5}
  [364] = {accel=80, decel=80, tmax=36.2, leave=0, reach=0.5}
  [365] = {accel=80, decel=80, tmax=38.504, leave=0, reach=0.5}
  [366] = {accel=80, decel=80, tmax=40.254, leave=0, reach=0.5}
  [367] = {accel=80, decel=80, tmax=41.256, leave=0, reach=0.5}
  [368] = {accel=80, decel=80, tmax=41.491, leave=0, reach=0.5}
  [369] = {accel=80, decel=80, tmax=41.066, leave=0, reach=0.5}
  [370] = {accel=80, decel=80, tmax=40.09, leave=0, reach=0.5}
  [371] = {accel=80, decel=80, tmax=38.629, leave=0, reach=0.5}
  [372] = {accel=80, decel=80, tmax=36.763, leave=0, reach=0.5}
  [373] = {accel=80, decel=80, tmax=34.628, leave=0, reach=0.5}
  [374] = {accel=80, decel=80, tmax=32.387, leave=0, reach=0.5}
  [375] = {accel=80, decel=80, tmax=30.176, leave=0, reach=0.5}
  [376] = {accel=80, decel=80, tmax=28.082, leave=0, reach=0.5}
  [377] = {accel=80, decel=80, tmax=26.155, leave=0, reach=0.5}
  [378] = {accel=80, decel=80, tmax=24.415, leave=0, reach=0.5}
  [379] = {accel=80, decel=80, tmax=22.855, leave=0, reach=0.5}
  [380] = {accel=80, decel=80, tmax=21.458, leave=0, reach=0.5}
  [381] = {accel=80, decel=80, tmax=20.206, leave=0, reach=0.5}
  [382] = {accel=80, decel=80, tmax=19.089, leave=0, reach=0.5}
  [383] = {accel=80, decel=80, tmax=18.1, leave=0, reach=0.5}
  [384] = {accel=80, decel=80, tmax=17.226, leave=0, reach=0.5}
  [385] = {accel=80, decel=80, tmax=16.45, leave=0, reach=0.5}
  [386] = {accel=80, decel=80, tmax=15.752, leave=0, reach=0.5}
  [387] = {accel=80, decel=80, tmax=15.113, leave=0, reach=0.5}
  [388] = {accel=80, decel=80, tmax=14.519, leave=0, reach=0.5}
  [389] = {accel=80, decel=80, tmax=14.009, leave=0, reach=0.5}
  [390] = {accel=80, decel=80, tmax=13.545, leave=0, reach=0.5}
  [391] = {accel=80, decel=80, tmax=13.06, leave=0, reach=0.5}
  [392] = {accel=80, decel=80, tmax=12.589, leave=0, reach=0.5}
  [393] = {accel=80, decel=80, tmax=12.162, leave=0, reach=0.5}
  [394] = {accel=80, decel=80, tmax=11.786, leave=0, reach=0.5}
  [395] = {accel=80, decel=80, tmax=11.467, leave=0, reach=0.5}
  [396] = {accel=80, decel=80, tmax=11.207, leave=0, reach=0.5}
  [397] = {accel=80, decel=80, tmax=11.009, leave=0, reach=0.5}
  [398] = {accel=80, decel=80, tmax=10.871, leave=0, reach=0.5}
  [399] = {accel=80, decel=80, tmax=10.791, leave=0, reach=0.5}
  [400] = {accel=80, decel=80, tmax=10.764, leave=0, reach=0.5}
  [401] = {accel=80, decel=80, tmax=10.779, leave=0, reach=0.5}
  [402] = {accel=80, decel=80, tmax=10.821, leave=0, reach=0.5}
  [403] = {accel=80, decel=80, tmax=10.871, leave=0, reach=0.5}
  [404] = {accel=80, decel=80, tmax=10.906, leave=0, reach=0.5}
  [405] = {accel=80, decel=80, tmax=10.913, leave=0, reach=0.5}
  [406] = {accel=80, decel=80, tmax=10.885, leave=0, reach=0.5}
  [407] = {accel=80, decel=80, tmax=10.815, leave=0, reach=0.5}
  [408] = {accel=80, decel=80, tmax=10.706, leave=0, reach=0.5}
  [409] = {accel=80, decel=80, tmax=10.572, leave=0, reach=0.5}
  [410] = {accel=80, decel=80, tmax=10.453, leave=0, reach=0.5}
  [411] = {accel=80, decel=80, tmax=10.388, leave=0, reach=0.5}
  [412] = {accel=80, decel=80, tmax=10.396, leave=0, reach=0.5}
  [413] = {accel=80, decel=80, tmax=10.457, leave=0, reach=0.5}
  [414] = {accel=80, decel=80, tmax=10.523, leave=0, reach=0.5}
  [415] = {accel=80, decel=80, tmax=10.549, leave=0, reach=0.5}
  [416] = {accel=80, decel=80, tmax=10.516, leave=0, reach=0.5}
  [417] = {accel=80, decel=80, tmax=10.44, leave=0, reach=0.5}
  [418] = {accel=80, decel=80, tmax=10.349, leave=0, reach=0.5}
  [419] = {accel=80, decel=80, tmax=10.267, leave=0, reach=0.5}
  [420] = {accel=80, decel=80, tmax=10.212, leave=0, reach=0.5}
  [421] = {accel=80, decel=80, tmax=10.185, leave=0, reach=0.5}
  [422] = {accel=80, decel=80, tmax=10.176, leave=0, reach=0.5}
  [423] = {accel=80, decel=80, tmax=10.172, leave=0, reach=0.5}
  [424] = {accel=80, decel=80, tmax=10.157, leave=0, reach=0.5}
  [425] = {accel=80, decel=80, tmax=10.124, leave=0, reach=0.5}
  [426] = {accel=80, decel=80, tmax=23.062, leave=0, reach=0.5}
  [427] = {accel=80, decel=80, tmax=10.578, leave=0, reach=0.5}
  [428] = {accel=80, decel=80, tmax=10.626, leave=0, reach=0.5}
  [429] = {accel=80, decel=80, tmax=10.655, leave=0, reach=0.5}
  [430] = {accel=80, decel=80, tmax=10.663, leave=0, reach=0.5}
  [431] = {accel=80, decel=80, tmax=10.654, leave=0, reach=0.5}
  [432] = {accel=80, decel=80, tmax=10.635, leave=0, reach=0.5}
  [433] = {accel=80, decel=80, tmax=10.62, leave=0, reach=0.5}
  [434] = {accel=80, decel=80, tmax=10.621, leave=0, reach=0.5}
  [435] = {accel=80, decel=80, tmax=10.649, leave=0, reach=0.5}
  [436] = {accel=80, decel=80, tmax=10.702, leave=0, reach=0.5}
  [437] = {accel=80, decel=80, tmax=10.767, leave=0, reach=0.5}
  [438] = {accel=80, decel=80, tmax=10.82, leave=0, reach=0.5}
  [439] = {accel=80, decel=80, tmax=10.835, leave=0, reach=0.5}
  [440] = {accel=80, decel=80, tmax=10.801, leave=0, reach=0.5}
  [441] = {accel=80, decel=80, tmax=10.735, leave=0, reach=0.5}
  [442] = {accel=80, decel=80, tmax=10.68, leave=0, reach=0.5}
  [443] = {accel=80, decel=80, tmax=10.675, leave=0, reach=0.5}
  [444] = {accel=80, decel=80, tmax=10.725, leave=0, reach=0.5}
  [445] = {accel=80, decel=80, tmax=10.808, leave=0, reach=0.5}
  [446] = {accel=80, decel=80, tmax=10.889, leave=0, reach=0.5}
  [447] = {accel=80, decel=80, tmax=10.945, leave=0, reach=0.5}
  [448] = {accel=80, decel=80, tmax=10.968, leave=0, reach=0.5}
  [449] = {accel=80, decel=80, tmax=10.963, leave=0, reach=0.5}
  [450] = {accel=80, decel=80, tmax=10.932, leave=0, reach=0.5}
  [451] = {accel=80, decel=80, tmax=10.877, leave=0, reach=0.5}
  [452] = {accel=80, decel=80, tmax=10.809, leave=0, reach=0.5}
  [453] = {accel=80, decel=80, tmax=10.744, leave=0, reach=0.5}
  [454] = {accel=80, decel=80, tmax=10.703, leave=0, reach=0.5}
  [455] = {accel=80, decel=80, tmax=10.702, leave=0, reach=0.5}
  [456] = {accel=80, decel=80, tmax=10.757, leave=0, reach=0.5}
  [457] = {accel=80, decel=80, tmax=10.878, leave=0, reach=0.5}
  [458] = {accel=80, decel=80, tmax=11.069, leave=0, reach=0.5}
  [459] = {accel=80, decel=80, tmax=11.33, leave=0, reach=0.5}
  [460] = {accel=80, decel=80, tmax=11.656, leave=0, reach=0.5}
  [461] = {accel=80, decel=80, tmax=12.039, leave=0, reach=0.5}
  [462] = {accel=80, decel=80, tmax=12.472, leave=0, reach=0.5}
  [463] = {accel=80, decel=80, tmax=12.95, leave=0, reach=0.5}
  [464] = {accel=80, decel=80, tmax=13.441, leave=0, reach=0.5}
  [465] = {accel=80, decel=80, tmax=13.909, leave=0, reach=0.5}
  [466] = {accel=80, decel=80, tmax=14.421, leave=0, reach=0.5}
  [467] = {accel=80, decel=80, tmax=15.011, leave=0, reach=0.5}
  [468] = {accel=80, decel=80, tmax=15.638, leave=0, reach=0.5}
  [469] = {accel=80, decel=80, tmax=16.319, leave=0, reach=0.5}
  [470] = {accel=80, decel=80, tmax=17.082, leave=0, reach=0.5}
  [471] = {accel=80, decel=80, tmax=17.954, leave=0, reach=0.5}
  [472] = {accel=80, decel=80, tmax=18.961, leave=0, reach=0.5}
  [473] = {accel=80, decel=80, tmax=20.118, leave=0, reach=0.5}
  [474] = {accel=80, decel=80, tmax=21.436, leave=0, reach=0.5}
  [475] = {accel=80, decel=80, tmax=22.92, leave=0, reach=0.5}
  [476] = {accel=80, decel=80, tmax=24.584, leave=0, reach=0.5}
  [477] = {accel=80, decel=80, tmax=26.449, leave=0, reach=0.5}
  [478] = {accel=80, decel=80, tmax=28.532, leave=0, reach=0.5}
  [479] = {accel=80, decel=80, tmax=30.828, leave=0, reach=0.5}
  [480] = {accel=80, decel=80, tmax=33.294, leave=0, reach=0.5}
  [481] = {accel=80, decel=80, tmax=35.842, leave=0, reach=0.5}
  [482] = {accel=80, decel=80, tmax=38.329, leave=0, reach=0.5}
  [483] = {accel=80, decel=80, tmax=40.579, leave=0, reach=0.5}
  [484] = {accel=80, decel=80, tmax=42.43, leave=0, reach=0.5}
  [485] = {accel=80, decel=80, tmax=43.768, leave=0, reach=0.5}
  [486] = {accel=80, decel=80, tmax=44.49, leave=0, reach=0.5}
  [487] = {accel=80, decel=80, tmax=44.462, leave=0, reach=0.5}
  [488] = {accel=80, decel=80, tmax=43.548, leave=0, reach=0.5}
  [489] = {accel=80, decel=80, tmax=41.744, leave=0, reach=0.5}
  [490] = {accel=80, decel=80, tmax=39.259, leave=0, reach=0.5}
  [491] = {accel=80, decel=80, tmax=36.427, leave=0, reach=0.5}
  [492] = {accel=80, decel=80, tmax=33.544, leave=0, reach=0.5}
  [493] = {accel=80, decel=80, tmax=30.787, leave=0, reach=0.5}
  [494] = {accel=80, decel=80, tmax=28.23, leave=0, reach=0.5}
  [495] = {accel=80, decel=80, tmax=25.881, leave=0, reach=0.5}
  [496] = {accel=80, decel=80, tmax=23.73, leave=0, reach=0.5}
  [497] = {accel=80, decel=80, tmax=21.767, leave=0, reach=0.5}
  [498] = {accel=80, decel=80, tmax=19.986, leave=0, reach=0.5}
  [499] = {accel=80, decel=80, tmax=18.384, leave=0, reach=0.5}
  [500] = {accel=80, decel=80, tmax=16.96, leave=0, reach=0.5}
  [501] = {accel=80, decel=80, tmax=15.704, leave=0, reach=0.5}
  [502] = {accel=80, decel=80, tmax=14.602, leave=0, reach=0.5}
  [503] = {accel=80, decel=80, tmax=30.805, leave=0, reach=0.5}
  [504] = {accel=80, decel=80, tmax=13.901, leave=0, reach=0.5}
  [505] = {accel=80, decel=80, tmax=14.804, leave=0, reach=0.5}
  [506] = {accel=80, decel=80, tmax=15.819, leave=0, reach=0.5}
  [507] = {accel=80, decel=80, tmax=16.982, leave=0, reach=0.5}
  [508] = {accel=80, decel=80, tmax=18.321, leave=0, reach=0.5}
  [509] = {accel=80, decel=80, tmax=19.85, leave=0, reach=0.5}
  [510] = {accel=80, decel=80, tmax=21.571, leave=0, reach=0.5}
  [511] = {accel=80, decel=80, tmax=23.478, leave=0, reach=0.5}
  [512] = {accel=80, decel=80, tmax=25.568, leave=0, reach=0.5}
  [513] = {accel=80, decel=80, tmax=27.846, leave=0, reach=0.5}
  [514] = {accel=80, decel=80, tmax=30.328, leave=0, reach=0.5}
  [515] = {accel=80, decel=80, tmax=33.028, leave=0, reach=0.5}
  [516] = {accel=80, decel=80, tmax=35.932, leave=0, reach=0.5}
  [517] = {accel=80, decel=80, tmax=38.957, leave=0, reach=0.5}
  [518] = {accel=80, decel=80, tmax=41.903, leave=0, reach=0.5}
  [519] = {accel=80, decel=80, tmax=44.441, leave=0, reach=0.5}
  [520] = {accel=80, decel=80, tmax=46.208, leave=0, reach=0.5}
  [521] = {accel=80, decel=80, tmax=46.981, leave=0, reach=0.5}
  [522] = {accel=80, decel=80, tmax=46.766, leave=0, reach=0.5}
  [523] = {accel=80, decel=80, tmax=45.717, leave=0, reach=0.5}
  [524] = {accel=80, decel=80, tmax=44.013, leave=0, reach=0.5}
  [525] = {accel=80, decel=80, tmax=41.813, leave=0, reach=0.5}
  [526] = {accel=80, decel=80, tmax=39.262, leave=0, reach=0.5}
  [527] = {accel=80, decel=80, tmax=36.52, leave=0, reach=0.5}
  [528] = {accel=80, decel=80, tmax=33.751, leave=0, reach=0.5}
  [529] = {accel=80, decel=80, tmax=31.094, leave=0, reach=0.5}
  [530] = {accel=80, decel=80, tmax=28.642, leave=0, reach=0.5}
  [531] = {accel=80, decel=80, tmax=26.437, leave=0, reach=0.5}
  [532] = {accel=80, decel=80, tmax=24.479, leave=0, reach=0.5}
  [533] = {accel=80, decel=80, tmax=22.743, leave=0, reach=0.5}
  [534] = {accel=80, decel=80, tmax=21.203, leave=0, reach=0.5}
  [535] = {accel=80, decel=80, tmax=19.848, leave=0, reach=0.5}
  [536] = {accel=80, decel=80, tmax=18.674, leave=0, reach=0.5}
  [537] = {accel=80, decel=80, tmax=17.671, leave=0, reach=0.5}
  [538] = {accel=80, decel=80, tmax=16.816, leave=0, reach=0.5}
  [539] = {accel=80, decel=80, tmax=16.078, leave=0, reach=0.5}
  [540] = {accel=80, decel=80, tmax=15.421, leave=0, reach=0.5}
  [541] = {accel=80, decel=80, tmax=14.812, leave=0, reach=0.5}
  [542] = {accel=80, decel=80, tmax=14.23, leave=0, reach=0.5}
  [543] = {accel=80, decel=80, tmax=13.721, leave=0, reach=0.5}
  [544] = {accel=80, decel=80, tmax=13.254, leave=0, reach=0.5}
  [545] = {accel=80, decel=80, tmax=12.763, leave=0, reach=0.5}
  [546] = {accel=80, decel=80, tmax=12.286, leave=0, reach=0.5}
  [547] = {accel=80, decel=80, tmax=11.854, leave=0, reach=0.5}
  [548] = {accel=80, decel=80, tmax=11.47, leave=0, reach=0.5}
  [549] = {accel=80, decel=80, tmax=11.142, leave=0, reach=0.5}
  [550] = {accel=80, decel=80, tmax=10.883, leave=0, reach=0.5}
  [551] = {accel=80, decel=80, tmax=10.701, leave=0, reach=0.5}
  [552] = {accel=80, decel=80, tmax=10.599, leave=0, reach=0.5}
  [553] = {accel=80, decel=80, tmax=10.568, leave=0, reach=0.5}
  [554] = {accel=80, decel=80, tmax=10.594, leave=0, reach=0.5}
  [555] = {accel=80, decel=80, tmax=10.657, leave=0, reach=0.5}
  [556] = {accel=80, decel=80, tmax=10.736, leave=0, reach=0.5}
  [557] = {accel=80, decel=80, tmax=10.813, leave=0, reach=0.5}
  [558] = {accel=80, decel=80, tmax=10.876, leave=0, reach=0.5}
  [559] = {accel=80, decel=80, tmax=10.922, leave=0, reach=0.5}
  [560] = {accel=80, decel=80, tmax=10.95, leave=0, reach=0.5}
  [561] = {accel=80, decel=80, tmax=10.961, leave=0, reach=0.5}
  [562] = {accel=80, decel=80, tmax=10.952, leave=0, reach=0.5}
  [563] = {accel=80, decel=80, tmax=10.924, leave=0, reach=0.5}
  [564] = {accel=80, decel=80, tmax=10.891, leave=0, reach=0.5}
  [565] = {accel=80, decel=80, tmax=10.876, leave=0, reach=0.5}
  [566] = {accel=80, decel=80, tmax=10.897, leave=0, reach=0.5}
  [567] = {accel=80, decel=80, tmax=10.953, leave=0, reach=0.5}
  [568] = {accel=80, decel=80, tmax=11.018, leave=0, reach=0.5}
  [569] = {accel=80, decel=80, tmax=11.059, leave=0, reach=0.5}
  [570] = {accel=80, decel=80, tmax=11.062, leave=0, reach=0.5}
  [571] = {accel=80, decel=80, tmax=11.037, leave=0, reach=0.5}
  [572] = {accel=80, decel=80, tmax=11.004, leave=0, reach=0.5}
  [573] = {accel=80, decel=80, tmax=10.983, leave=0, reach=0.5}
  [574] = {accel=80, decel=80, tmax=10.985, leave=0, reach=0.5}
  [575] = {accel=80, decel=80, tmax=11.01, leave=0, reach=0.5}
  [576] = {accel=80, decel=80, tmax=11.05, leave=0, reach=0.5}
  [577] = {accel=80, decel=80, tmax=11.094, leave=0, reach=0.5}
  [578] = {accel=80, decel=80, tmax=11.13, leave=0, reach=0.5}
  [579] = {accel=80, decel=80, tmax=11.151, leave=0, reach=0.5}
  [580] = {accel=80, decel=80, tmax=11.152, leave=0, reach=0.5}
  [581] = {accel=80, decel=80, tmax=11.131, leave=0, reach=0.5}
  [582] = {accel=80, decel=80, tmax=11.083, leave=0, reach=0.5}
  [583] = {accel=80, decel=80, tmax=11.008, leave=0, reach=0.5}
  [584] = {accel=80, decel=80, tmax=24.885, leave=0, reach=0.5}
  [585] = {accel=80, decel=80, tmax=11.379, leave=0, reach=0.5}
  [586] = {accel=80, decel=80, tmax=11.489, leave=0, reach=0.5}
  [587] = {accel=80, decel=80, tmax=11.574, leave=0, reach=0.5}
  [588] = {accel=80, decel=80, tmax=11.628, leave=0, reach=0.5}
  [589] = {accel=80, decel=80, tmax=11.648, leave=0, reach=0.5}
  [590] = {accel=80, decel=80, tmax=11.635, leave=0, reach=0.5}
  [591] = {accel=80, decel=80, tmax=11.597, leave=0, reach=0.5}
  [592] = {accel=80, decel=80, tmax=11.541, leave=0, reach=0.5}
  [593] = {accel=80, decel=80, tmax=11.475, leave=0, reach=0.5}
  [594] = {accel=80, decel=80, tmax=11.405, leave=0, reach=0.5}
  [595] = {accel=80, decel=80, tmax=11.342, leave=0, reach=0.5}
  [596] = {accel=80, decel=80, tmax=11.292, leave=0, reach=0.5}
  [597] = {accel=80, decel=80, tmax=11.26, leave=0, reach=0.5}
  [598] = {accel=80, decel=80, tmax=11.246, leave=0, reach=0.5}
  [599] = {accel=80, decel=80, tmax=11.242, leave=0, reach=0.5}
  [600] = {accel=80, decel=80, tmax=11.234, leave=0, reach=0.5}
  [601] = {accel=80, decel=80, tmax=11.203, leave=0, reach=0.5}
  [602] = {accel=80, decel=80, tmax=11.142, leave=0, reach=0.5}
  [603] = {accel=80, decel=80, tmax=11.06, leave=0, reach=0.5}
  [604] = {accel=80, decel=80, tmax=10.982, leave=0, reach=0.5}
  [605] = {accel=80, decel=80, tmax=10.928, leave=0, reach=0.5}
  [606] = {accel=80, decel=80, tmax=10.902, leave=0, reach=0.5}
  [607] = {accel=80, decel=80, tmax=10.893, leave=0, reach=0.5}
  [608] = {accel=80, decel=80, tmax=10.886, leave=0, reach=0.5}
  [609] = {accel=80, decel=80, tmax=10.869, leave=0, reach=0.5}
  [610] = {accel=80, decel=80, tmax=10.84, leave=0, reach=0.5}
  [611] = {accel=80, decel=80, tmax=10.801, leave=0, reach=0.5}
  [612] = {accel=80, decel=80, tmax=10.753, leave=0, reach=0.5}
  [613] = {accel=80, decel=80, tmax=10.69, leave=0, reach=0.5}
  [614] = {accel=80, decel=80, tmax=10.613, leave=0, reach=0.5}
  [615] = {accel=80, decel=80, tmax=10.528, leave=0, reach=0.5}
  [616] = {accel=80, decel=80, tmax=10.452, leave=0, reach=0.5}
  [617] = {accel=80, decel=80, tmax=10.406, leave=0, reach=0.5}
  [618] = {accel=80, decel=80, tmax=10.415, leave=0, reach=0.5}
  [619] = {accel=80, decel=80, tmax=10.5, leave=0, reach=0.5}
  [620] = {accel=80, decel=80, tmax=10.67, leave=0, reach=0.5}
  [621] = {accel=80, decel=80, tmax=10.923, leave=0, reach=0.5}
  [622] = {accel=80, decel=80, tmax=11.246, leave=0, reach=0.5}
  [623] = {accel=80, decel=80, tmax=11.626, leave=0, reach=0.5}
  [624] = {accel=80, decel=80, tmax=12.051, leave=0, reach=0.5}
  [625] = {accel=80, decel=80, tmax=12.52, leave=0, reach=0.5}
  [626] = {accel=80, decel=80, tmax=13.004, leave=0, reach=0.5}
  [627] = {accel=80, decel=80, tmax=13.465, leave=0, reach=0.5}
  [628] = {accel=80, decel=80, tmax=13.967, leave=0, reach=0.5}
  [629] = {accel=80, decel=80, tmax=14.537, leave=0, reach=0.5}
  [630] = {accel=80, decel=80, tmax=15.127, leave=0, reach=0.5}
  [631] = {accel=80, decel=80, tmax=15.758, leave=0, reach=0.5}
  [632] = {accel=80, decel=80, tmax=16.468, leave=0, reach=0.5}
  [633] = {accel=80, decel=80, tmax=17.296, leave=0, reach=0.5}
  [634] = {accel=80, decel=80, tmax=18.282, leave=0, reach=0.5}
  [635] = {accel=80, decel=80, tmax=19.45, leave=0, reach=0.5}
  [636] = {accel=80, decel=80, tmax=20.812, leave=0, reach=0.5}
  [637] = {accel=80, decel=80, tmax=22.374, leave=0, reach=0.5}
  [638] = {accel=80, decel=80, tmax=24.148, leave=0, reach=0.5}
  [639] = {accel=80, decel=80, tmax=26.164, leave=0, reach=0.5}
  [640] = {accel=80, decel=80, tmax=28.449, leave=0, reach=0.5}
  [641] = {accel=80, decel=80, tmax=31.002, leave=0, reach=0.5}
  [642] = {accel=80, decel=80, tmax=33.769, leave=0, reach=0.5}
  [643] = {accel=80, decel=80, tmax=36.649, leave=0, reach=0.5}
  [644] = {accel=80, decel=80, tmax=39.51, leave=0, reach=0.5}
  [645] = {accel=80, decel=80, tmax=42.215, leave=0, reach=0.5}
  [646] = {accel=80, decel=80, tmax=44.64, leave=0, reach=0.5}
  [647] = {accel=80, decel=80, tmax=46.638, leave=0, reach=0.5}
  [648] = {accel=80, decel=80, tmax=48.009, leave=0, reach=0.5}
  [649] = {accel=80, decel=80, tmax=48.517, leave=0, reach=0.5}
  [650] = {accel=80, decel=80, tmax=47.981, leave=0, reach=0.5}
  [651] = {accel=80, decel=80, tmax=46.394, leave=0, reach=0.5}
  [652] = {accel=80, decel=80, tmax=43.975, leave=0, reach=0.5}
  [653] = {accel=80, decel=80, tmax=41.079, leave=0, reach=0.5}
  [654] = {accel=80, decel=80, tmax=38.035, leave=0, reach=0.5}
  [655] = {accel=80, decel=80, tmax=35.06, leave=0, reach=0.5}
  [656] = {accel=80, decel=80, tmax=32.255, leave=0, reach=0.5}
  [657] = {accel=80, decel=80, tmax=29.651, leave=0, reach=0.5}
  [658] = {accel=80, decel=80, tmax=27.245, leave=0, reach=0.5}
  [659] = {accel=80, decel=80, tmax=25.029, leave=0, reach=0.5}
  [660] = {accel=80, decel=80, tmax=23, leave=0, reach=0.5}
  [661] = {accel=80, decel=80, tmax=21.168, leave=0, reach=0.5}
  [662] = {accel=80, decel=80, tmax=19.55, leave=0, reach=0.5}
  [663] = {accel=80, decel=80, tmax=18.15, leave=0, reach=0.5}
  [664] = {accel=80, decel=80, tmax=16.952, leave=0, reach=0.5}
  [665] = {accel=80, decel=80, tmax=15.921, leave=0, reach=0.5}
  [666] = {accel=80, decel=80, tmax=15.013, leave=0, reach=0.5}
  [667] = {accel=80, decel=80, tmax=14.187, leave=0, reach=0.5}
  [668] = {accel=80, decel=80, tmax=13.413, leave=0, reach=0.5}
  [669] = {accel=80, decel=80, tmax=18.717, leave=0, reach=0.5}
  [670] = {accel=80, decel=80, tmax=13.798, leave=0, reach=0.5}
  [671] = {accel=80, decel=80, tmax=14.523, leave=0, reach=0.5}
  [672] = {accel=80, decel=80, tmax=15.274, leave=0, reach=0.5}
  [673] = {accel=80, decel=80, tmax=16.074, leave=0, reach=0.5}
  [674] = {accel=80, decel=80, tmax=16.958, leave=0, reach=0.5}
  [675] = {accel=80, decel=80, tmax=17.974, leave=0, reach=0.5}
  [676] = {accel=80, decel=80, tmax=19.175, leave=0, reach=0.5}
  [677] = {accel=80, decel=80, tmax=20.605, leave=0, reach=0.5}
  [678] = {accel=80, decel=80, tmax=22.281, leave=0, reach=0.5}
  [679] = {accel=80, decel=80, tmax=24.192, leave=0, reach=0.5}
  [680] = {accel=80, decel=80, tmax=26.308, leave=0, reach=0.5}
  [681] = {accel=80, decel=80, tmax=28.611, leave=0, reach=0.5}
  [682] = {accel=80, decel=80, tmax=31.096, leave=0, reach=0.5}
  [683] = {accel=80, decel=80, tmax=33.765, leave=0, reach=0.5}
  [684] = {accel=80, decel=80, tmax=36.603, leave=0, reach=0.5}
  [685] = {accel=80, decel=80, tmax=39.556, leave=0, reach=0.5}
  [686] = {accel=80, decel=80, tmax=42.507, leave=0, reach=0.5}
  [687] = {accel=80, decel=80, tmax=45.231, leave=0, reach=0.5}
  [688] = {accel=80, decel=80, tmax=47.408, leave=0, reach=0.5}
  [689] = {accel=80, decel=80, tmax=48.705, leave=0, reach=0.5}
  [690] = {accel=80, decel=80, tmax=48.929, leave=0, reach=0.5}
  [691] = {accel=80, decel=80, tmax=48.119, leave=0, reach=0.5}
  [692] = {accel=80, decel=80, tmax=46.496, leave=0, reach=0.5}
  [693] = {accel=80, decel=80, tmax=44.328, leave=0, reach=0.5}
  [694] = {accel=80, decel=80, tmax=41.826, leave=0, reach=0.5}
  [695] = {accel=80, decel=80, tmax=39.104, leave=0, reach=0.5}
  [696] = {accel=80, decel=80, tmax=36.247, leave=0, reach=0.5}
  [697] = {accel=80, decel=80, tmax=33.359, leave=0, reach=0.5}
  [698] = {accel=80, decel=80, tmax=30.564, leave=0, reach=0.5}
  [699] = {accel=80, decel=80, tmax=27.975, leave=0, reach=0.5}
  [700] = {accel=80, decel=80, tmax=25.657, leave=0, reach=0.5}
  [701] = {accel=80, decel=80, tmax=23.623, leave=0, reach=0.5}
  [702] = {accel=80, decel=80, tmax=21.848, leave=0, reach=0.5}
  [703] = {accel=80, decel=80, tmax=20.299, leave=0, reach=0.5}
  [704] = {accel=80, decel=80, tmax=18.958, leave=0, reach=0.5}
  [705] = {accel=80, decel=80, tmax=17.818, leave=0, reach=0.5}
  [706] = {accel=80, decel=80, tmax=16.862, leave=0, reach=0.5}
  [707] = {accel=80, decel=80, tmax=16.062, leave=0, reach=0.5}
  [708] = {accel=80, decel=80, tmax=15.38, leave=0, reach=0.5}
  [709] = {accel=80, decel=80, tmax=14.77, leave=0, reach=0.5}
  [710] = {accel=80, decel=80, tmax=14.197, leave=0, reach=0.5}
  [711] = {accel=80, decel=80, tmax=13.641, leave=0, reach=0.5}
  [712] = {accel=80, decel=80, tmax=13.152, leave=0, reach=0.5}
  [713] = {accel=80, decel=80, tmax=12.703, leave=0, reach=0.5}
  [714] = {accel=80, decel=80, tmax=12.233, leave=0, reach=0.5}
  [715] = {accel=80, decel=80, tmax=11.779, leave=0, reach=0.5}
  [716] = {accel=80, decel=80, tmax=11.367, leave=0, reach=0.5}
  [717] = {accel=80, decel=80, tmax=11, leave=0, reach=0.5}
  [718] = {accel=80, decel=80, tmax=10.688, leave=0, reach=0.5}
  [719] = {accel=80, decel=80, tmax=10.447, leave=0, reach=0.5}
  [720] = {accel=80, decel=80, tmax=10.291, leave=0, reach=0.5}
  [721] = {accel=80, decel=80, tmax=10.221, leave=0, reach=0.5}
  [722] = {accel=80, decel=80, tmax=10.227, leave=0, reach=0.5}
  [723] = {accel=80, decel=80, tmax=10.284, leave=0, reach=0.5}
  [724] = {accel=80, decel=80, tmax=10.366, leave=0, reach=0.5}
  [725] = {accel=80, decel=80, tmax=10.449, leave=0, reach=0.5}
  [726] = {accel=80, decel=80, tmax=10.521, leave=0, reach=0.5}
  [727] = {accel=80, decel=80, tmax=10.578, leave=0, reach=0.5}
  [728] = {accel=80, decel=80, tmax=10.624, leave=0, reach=0.5}
  [729] = {accel=80, decel=80, tmax=10.663, leave=0, reach=0.5}
  [730] = {accel=80, decel=80, tmax=10.696, leave=0, reach=0.5}
  [731] = {accel=80, decel=80, tmax=10.72, leave=0, reach=0.5}
  [732] = {accel=80, decel=80, tmax=10.741, leave=0, reach=0.5}
  [733] = {accel=80, decel=80, tmax=10.773, leave=0, reach=0.5}
  [734] = {accel=80, decel=80, tmax=10.833, leave=0, reach=0.5}
  [735] = {accel=80, decel=80, tmax=10.925, leave=0, reach=0.5}
  [736] = {accel=80, decel=80, tmax=11.042, leave=0, reach=0.5}
  [737] = {accel=80, decel=80, tmax=11.158, leave=0, reach=0.5}
  [738] = {accel=80, decel=80, tmax=11.254, leave=0, reach=0.5}
  [739] = {accel=80, decel=80, tmax=11.32, leave=0, reach=0.5}
  [740] = {accel=80, decel=80, tmax=11.367, leave=0, reach=0.5}
  [741] = {accel=80, decel=80, tmax=11.407, leave=0, reach=0.5}
  [742] = {accel=80, decel=80, tmax=11.455, leave=0, reach=0.5}
  [743] = {accel=80, decel=80, tmax=11.516, leave=0, reach=0.5}
  [744] = {accel=80, decel=80, tmax=11.59, leave=0, reach=0.5}
  [745] = {accel=80, decel=80, tmax=11.678, leave=0, reach=0.5}
  [746] = {accel=80, decel=80, tmax=11.776, leave=0, reach=0.5}
  [747] = {accel=80, decel=80, tmax=11.878, leave=0, reach=0.5}
  [748] = {accel=80, decel=80, tmax=11.976, leave=0, reach=0.5}
  [749] = {accel=80, decel=80, tmax=12.059, leave=0, reach=0.5}
  [750] = {accel=80, decel=80, tmax=12.114, leave=0, reach=0.5}
  [751] = {accel=80, decel=80, tmax=12.134, leave=0, reach=0.5}
  [752] = {accel=80, decel=80, tmax=12.114, leave=0, reach=0.5}
  [753] = {accel=80, decel=80, tmax=12.059, leave=0, reach=0.5}
  [754] = {accel=80, decel=80, tmax=11.978, leave=0, reach=0.5}
  [755] = {accel=80, decel=80, tmax=11.876, leave=0, reach=0.5}
  [756] = {accel=80, decel=80, tmax=11.753, leave=0, reach=0.5}
  [757] = {accel=80, decel=80, tmax=26.478, leave=0, reach=0.5}
  [758] = {accel=80, decel=80, tmax=12.123, leave=0, reach=0.5}
  [759] = {accel=80, decel=80, tmax=12.29, leave=0, reach=0.5}
  [760] = {accel=80, decel=80, tmax=12.413, leave=0, reach=0.5}
  [761] = {accel=80, decel=80, tmax=12.502, leave=0, reach=0.5}
  [762] = {accel=80, decel=80, tmax=12.565, leave=0, reach=0.5}
  [763] = {accel=80, decel=80, tmax=12.604, leave=0, reach=0.5}
  [764] = {accel=80, decel=80, tmax=12.613, leave=0, reach=0.5}
  [765] = {accel=80, decel=80, tmax=12.583, leave=0, reach=0.5}
  [766] = {accel=80, decel=80, tmax=12.512, leave=0, reach=0.5}
  [767] = {accel=80, decel=80, tmax=12.403, leave=0, reach=0.5}
  [768] = {accel=80, decel=80, tmax=12.269, leave=0, reach=0.5}
  [769] = {accel=80, decel=80, tmax=12.124, leave=0, reach=0.5}
  [770] = {accel=80, decel=80, tmax=11.98, leave=0, reach=0.5}
  [771] = {accel=80, decel=80, tmax=11.849, leave=0, reach=0.5}
  [772] = {accel=80, decel=80, tmax=11.733, leave=0, reach=0.5}
  [773] = {accel=80, decel=80, tmax=11.633, leave=0, reach=0.5}
  [774] = {accel=80, decel=80, tmax=11.546, leave=0, reach=0.5}
  [775] = {accel=80, decel=80, tmax=11.469, leave=0, reach=0.5}
  [776] = {accel=80, decel=80, tmax=11.397, leave=0, reach=0.5}
  [777] = {accel=80, decel=80, tmax=11.317, leave=0, reach=0.5}
  [778] = {accel=80, decel=80, tmax=11.215, leave=0, reach=0.5}
  [779] = {accel=80, decel=80, tmax=11.081, leave=0, reach=0.5}
  [780] = {accel=80, decel=80, tmax=10.923, leave=0, reach=0.5}
  [781] = {accel=80, decel=80, tmax=10.767, leave=0, reach=0.5}
  [782] = {accel=80, decel=80, tmax=10.641, leave=0, reach=0.5}
  [783] = {accel=80, decel=80, tmax=10.559, leave=0, reach=0.5}
  [784] = {accel=80, decel=80, tmax=10.516, leave=0, reach=0.5}
  [785] = {accel=80, decel=80, tmax=10.493, leave=0, reach=0.5}
  [786] = {accel=80, decel=80, tmax=10.472, leave=0, reach=0.5}
  [787] = {accel=80, decel=80, tmax=10.444, leave=0, reach=0.5}
  [788] = {accel=80, decel=80, tmax=10.409, leave=0, reach=0.5}
  [789] = {accel=80, decel=80, tmax=10.368, leave=0, reach=0.5}
  [790] = {accel=80, decel=80, tmax=10.318, leave=0, reach=0.5}
  [791] = {accel=80, decel=80, tmax=10.254, leave=0, reach=0.5}
  [792] = {accel=80, decel=80, tmax=10.177, leave=0, reach=0.5}
  [793] = {accel=80, decel=80, tmax=10.098, leave=0, reach=0.5}
  [794] = {accel=80, decel=80, tmax=10.037, leave=0, reach=0.5}
  [795] = {accel=80, decel=80, tmax=10.023, leave=0, reach=0.5}
  [796] = {accel=80, decel=80, tmax=10.081, leave=0, reach=0.5}
  [797] = {accel=80, decel=80, tmax=10.222, leave=0, reach=0.5}
  [798] = {accel=80, decel=80, tmax=10.445, leave=0, reach=0.5}
  [799] = {accel=80, decel=80, tmax=10.739, leave=0, reach=0.5}
  [800] = {accel=80, decel=80, tmax=11.087, leave=0, reach=0.5}
  [801] = {accel=80, decel=80, tmax=11.479, leave=0, reach=0.5}
  [802] = {accel=80, decel=80, tmax=11.911, leave=0, reach=0.5}
  [803] = {accel=80, decel=80, tmax=12.359, leave=0, reach=0.5}
  [804] = {accel=80, decel=80, tmax=12.789, leave=0, reach=0.5}
  [805] = {accel=80, decel=80, tmax=13.262, leave=0, reach=0.5}
  [806] = {accel=80, decel=80, tmax=13.803, leave=0, reach=0.5}
  [807] = {accel=80, decel=80, tmax=14.362, leave=0, reach=0.5}
  [808] = {accel=80, decel=80, tmax=14.954, leave=0, reach=0.5}
  [809] = {accel=80, decel=80, tmax=15.612, leave=0, reach=0.5}
  [810] = {accel=80, decel=80, tmax=16.379, leave=0, reach=0.5}
  [811] = {accel=80, decel=80, tmax=17.295, leave=0, reach=0.5}
  [812] = {accel=80, decel=80, tmax=18.389, leave=0, reach=0.5}
  [813] = {accel=80, decel=80, tmax=19.678, leave=0, reach=0.5}
  [814] = {accel=80, decel=80, tmax=21.179, leave=0, reach=0.5}
  [815] = {accel=80, decel=80, tmax=22.917, leave=0, reach=0.5}
  [816] = {accel=80, decel=80, tmax=24.925, leave=0, reach=0.5}
  [817] = {accel=80, decel=80, tmax=27.221, leave=0, reach=0.5}
  [818] = {accel=80, decel=80, tmax=29.778, leave=0, reach=0.5}
  [819] = {accel=80, decel=80, tmax=32.519, leave=0, reach=0.5}
  [820] = {accel=80, decel=80, tmax=35.33, leave=0, reach=0.5}
  [821] = {accel=80, decel=80, tmax=38.098, leave=0, reach=0.5}
  [822] = {accel=80, decel=80, tmax=40.744, leave=0, reach=0.5}
  [823] = {accel=80, decel=80, tmax=43.22, leave=0, reach=0.5}
  [824] = {accel=80, decel=80, tmax=45.441, leave=0, reach=0.5}
  [825] = {accel=80, decel=80, tmax=47.219, leave=0, reach=0.5}
  [826] = {accel=80, decel=80, tmax=48.283, leave=0, reach=0.5}
  [827] = {accel=80, decel=80, tmax=48.374, leave=0, reach=0.5}
  [828] = {accel=80, decel=80, tmax=47.399, leave=0, reach=0.5}
  [829] = {accel=80, decel=80, tmax=45.505, leave=0, reach=0.5}
  [830] = {accel=80, decel=80, tmax=43.001, leave=0, reach=0.5}
  [831] = {accel=80, decel=80, tmax=40.21, leave=0, reach=0.5}
  [832] = {accel=80, decel=80, tmax=37.364, leave=0, reach=0.5}
  [833] = {accel=80, decel=80, tmax=34.6, leave=0, reach=0.5}
  [834] = {accel=80, decel=80, tmax=31.977, leave=0, reach=0.5}
  [835] = {accel=80, decel=80, tmax=29.517, leave=0, reach=0.5}
  [836] = {accel=80, decel=80, tmax=27.222, leave=0, reach=0.5}
  [837] = {accel=80, decel=80, tmax=25.099, leave=0, reach=0.5}
  [838] = {accel=80, decel=80, tmax=23.178, leave=0, reach=0.5}
  [839] = {accel=80, decel=80, tmax=21.497, leave=0, reach=0.5}
  [840] = {accel=80, decel=80, tmax=20.076, leave=0, reach=0.5}
  [841] = {accel=80, decel=80, tmax=18.898, leave=0, reach=0.5}
  [842] = {accel=80, decel=80, tmax=17.917, leave=0, reach=0.5}
  [843] = {accel=80, decel=80, tmax=17.076, leave=0, reach=0.5}
  [844] = {accel=80, decel=80, tmax=16.322, leave=0, reach=0.5}
  [845] = {accel=80, decel=80, tmax=15.615, leave=0, reach=0.5}
  [846] = {accel=80, decel=80, tmax=14.929, leave=0, reach=0.5}
  [847] = {accel=80, decel=80, tmax=14.239, leave=0, reach=0.5}
  [848] = {accel=80, decel=80, tmax=13.531, leave=0, reach=0.5}
  [849] = {accel=80, decel=80, tmax=29.038, leave=0, reach=0.5}
  [850] = {accel=80, decel=80, tmax=13.204, leave=0, reach=0.5}
  [851] = {accel=80, decel=80, tmax=13.971, leave=0, reach=0.5}
  [852] = {accel=80, decel=80, tmax=14.698, leave=0, reach=0.5}
  [853] = {accel=80, decel=80, tmax=15.378, leave=0, reach=0.5}
  [854] = {accel=80, decel=80, tmax=16.022, leave=0, reach=0.5}
  [855] = {accel=80, decel=80, tmax=16.655, leave=0, reach=0.5}
  [856] = {accel=80, decel=80, tmax=17.306, leave=0, reach=0.5}
  [857] = {accel=80, decel=80, tmax=18.008, leave=0, reach=0.5}
  [858] = {accel=80, decel=80, tmax=18.803, leave=0, reach=0.5}
  [859] = {accel=80, decel=80, tmax=19.739, leave=0, reach=0.5}
  [860] = {accel=80, decel=80, tmax=20.87, leave=0, reach=0.5}
  [861] = {accel=80, decel=80, tmax=22.236, leave=0, reach=0.5}
  [862] = {accel=80, decel=80, tmax=23.85, leave=0, reach=0.5}
  [863] = {accel=80, decel=80, tmax=25.687, leave=0, reach=0.5}
  [864] = {accel=80, decel=80, tmax=27.708, leave=0, reach=0.5}
  [865] = {accel=80, decel=80, tmax=29.879, leave=0, reach=0.5}
  [866] = {accel=80, decel=80, tmax=32.196, leave=0, reach=0.5}
  [867] = {accel=80, decel=80, tmax=34.662, leave=0, reach=0.5}
  [868] = {accel=80, decel=80, tmax=37.265, leave=0, reach=0.5}
  [869] = {accel=80, decel=80, tmax=39.947, leave=0, reach=0.5}
  [870] = {accel=80, decel=80, tmax=42.557, leave=0, reach=0.5}
  [871] = {accel=80, decel=80, tmax=44.836, leave=0, reach=0.5}
  [872] = {accel=80, decel=80, tmax=46.453, leave=0, reach=0.5}
  [873] = {accel=80, decel=80, tmax=47.127, leave=0, reach=0.5}
  [874] = {accel=80, decel=80, tmax=46.769, leave=0, reach=0.5}
  [875] = {accel=80, decel=80, tmax=45.526, leave=0, reach=0.5}
  [876] = {accel=80, decel=80, tmax=43.678, leave=0, reach=0.5}
  [877] = {accel=80, decel=80, tmax=41.479, leave=0, reach=0.5}
  [878] = {accel=80, decel=80, tmax=39.086, leave=0, reach=0.5}
  [879] = {accel=80, decel=80, tmax=36.561, leave=0, reach=0.5}
  [880] = {accel=80, decel=80, tmax=33.935, leave=0, reach=0.5}
  [881] = {accel=80, decel=80, tmax=31.267, leave=0, reach=0.5}
  [882] = {accel=80, decel=80, tmax=28.651, leave=0, reach=0.5}
  [883] = {accel=80, decel=80, tmax=26.193, leave=0, reach=0.5}
  [884] = {accel=80, decel=80, tmax=23.976, leave=0, reach=0.5}
  [885] = {accel=80, decel=80, tmax=22.038, leave=0, reach=0.5}
  [886] = {accel=80, decel=80, tmax=20.372, leave=0, reach=0.5}
  [887] = {accel=80, decel=80, tmax=18.95, leave=0, reach=0.5}
  [888] = {accel=80, decel=80, tmax=17.736, leave=0, reach=0.5}
  [889] = {accel=80, decel=80, tmax=16.707, leave=0, reach=0.5}
  [890] = {accel=80, decel=80, tmax=15.843, leave=0, reach=0.5}
  [891] = {accel=80, decel=80, tmax=15.114, leave=0, reach=0.5}
  [892] = {accel=80, decel=80, tmax=14.482, leave=0, reach=0.5}
  [893] = {accel=80, decel=80, tmax=13.907, leave=0, reach=0.5}
  [894] = {accel=80, decel=80, tmax=13.363, leave=0, reach=0.5}
  [895] = {accel=80, decel=80, tmax=12.84, leave=0, reach=0.5}
  [896] = {accel=80, decel=80, tmax=12.389, leave=0, reach=0.5}
  [897] = {accel=80, decel=80, tmax=11.984, leave=0, reach=0.5}
  [898] = {accel=80, decel=80, tmax=11.563, leave=0, reach=0.5}
  [899] = {accel=80, decel=80, tmax=11.157, leave=0, reach=0.5}
  [900] = {accel=80, decel=80, tmax=10.791, leave=0, reach=0.5}
  [901] = {accel=80, decel=80, tmax=10.468, leave=0, reach=0.5}
  [902] = {accel=30, decel=30, tmax=100, leave=0, reach=0.5}
  [903] = {accel=30, decel=30, tmax=100, leave=0, reach=0.5}
  [904] = {accel=30, decel=30, tmax=100, leave=0, reach=0.5}
  [905] = {accel=30, decel=30, tmax=100, leave=0, reach=0.5}
  [906] = {accel=30, decel=30, tmax=100, leave=0, reach=0.5}
  [907] = {accel=30, decel=30, tmax=100, leave=0, reach=0.5}
  [908] = {accel=30, decel=30, tmax=100, leave=0, reach=0.5}
  [909] = {accel=30, decel=30, tmax=100, leave=0, reach=0.5}
  [910] = {accel=30, decel=30, tmax=100, leave=0, reach=0.5}
  [911] = {accel=30, decel=30, tmax=100, leave=0, reach=0.5}
  [912] = {accel=30, decel=30, tmax=100, leave=0, reach=0.5}
  [913] = {accel=30, decel=30, tmax=100, leave=0, reach=0.5}
  [914] = {accel=30, decel=30, tmax=100, leave=0, reach=0.5}
  [915] = {accel=30, decel=30, tmax=100, leave=0, reach=0.5}
  [916] = {accel=30, decel=30, tmax=100, leave=0, reach=0.5}
  [917] = {accel=30, decel=30, tmax=100, leave=0, reach=0.5}
  [918] = {accel=30, decel=30, tmax=100, leave=0, reach=0.5}
  [919] = {accel=30, decel=30, tmax=100, leave=0, reach=0.5}
  [920] = {accel=30, decel=30, tmax=100, leave=0, reach=0.5}
  [921] = {accel=30, decel=30, tmax=100, leave=0, reach=0.5}
  [922] = {accel=30, decel=30, tmax=100, leave=0, reach=0.5}
  [923] = {accel=30, decel=30, tmax=100, leave=0, reach=0.5}
  [924] = {accel=30, decel=30, tmax=100, leave=0, reach=0.5}
  [925] = {accel=30, decel=30, tmax=100, leave=0, reach=0.5}
  [926] = {accel=30, decel=30, tmax=100, leave=0, reach=0.5}
  [927] = {accel=30, decel=30, tmax=100, leave=0, reach=0.5}
  [928] = {accel=30, decel=30, tmax=100, leave=0, reach=0.5}
  [929] = {accel=30, decel=30, tmax=100, leave=0, reach=0.5}
  [930] = {accel=30, decel=30, tmax=100, leave=0, reach=0.5}
  [931] = {accel=30, decel=30, tmax=100, leave=0, reach=0.5}
  [932] = {accel=30, decel=30, tmax=100, leave=0, reach=0.5}
  [933] = {accel=30, decel=30, tmax=100, leave=0, reach=0.5}
  [934] = {accel=30, decel=30, tmax=100, leave=0, reach=0.5}
  [935] = {accel=30, decel=30, tmax=100, leave=0, reach=0.5}
  [936] = {accel=30, decel=30, tmax=100, leave=0, reach=0.5}
  [937] = {accel=30, decel=30, tmax=100, leave=0, reach=0.5}
  [938] = {accel=30, decel=30, tmax=100, leave=0, reach=0.5}
  [939] = {accel=30, decel=30, tmax=100, leave=0, reach=0.5}
  [940] = {accel=30, decel=30, tmax=100, leave=0, reach=0.5}
  [941] = {accel=30, decel=30, tmax=100, leave=0, reach=0.5}
  [942] = {accel=30, decel=30, tmax=100, leave=0, reach=0.5}
  [943] = {accel=30, decel=30, tmax=100, leave=0, reach=0.5}
  [944] = {accel=30, decel=30, tmax=100, leave=0, reach=0.5}
  [945] = {accel=30, decel=30, tmax=100, leave=0, reach=0.5}
  [946] = {accel=30, decel=30, tmax=100, leave=0, reach=0.5}
  [947] = {accel=30, decel=30, tmax=100, leave=0, reach=0.5}
  [948] = {accel=30, decel=30, tmax=100, leave=0, reach=0.5}
  [949] = {accel=30, decel=30, tmax=100, leave=0, reach=0.5}
  [950] = {accel=30, decel=30, tmax=100, leave=0, reach=0.5}
  [951] = {accel=30, decel=30, tmax=100, leave=0, reach=0.5}
  [952] = {accel=30, decel=30, tmax=100, leave=0, reach=0.5}
  [953] = {accel=30, decel=30, tmax=100, leave=0, reach=0.5}
  [954] = {accel=30, decel=30, tmax=100, leave=0, reach=0.5}
  [955] = {accel=30, decel=30, tmax=100, leave=0, reach=0.5}
  [956] = {accel=30, decel=30, tmax=100, leave=0, reach=0.5}
  [957] = {accel=30, decel=30, tmax=100, leave=0, reach=0.5}
  [958] = {accel=30, decel=30, tmax=100, leave=0, reach=0.5}
  [959] = {accel=30, decel=30, tmax=100, leave=0, reach=0.5}
  [960] = {accel=30, decel=30, tmax=100, leave=0, reach=0.5}
  [961] = {accel=30, decel=30, tmax=100, leave=0, reach=0.5}
  [962] = {accel=30, decel=30, tmax=100, leave=0, reach=0.5}
  [963] = {accel=30, decel=30, tmax=100, leave=0, reach=0.5}
  [964] = {accel=30, decel=30, tmax=100, leave=0, reach=0.5}
  [965] = {accel=30, decel=30, tmax=100, leave=0, reach=0.5}
  [966] = {accel=30, decel=30, tmax=100, leave=0, reach=0.5}
  [967] = {accel=30, decel=30, tmax=100, leave=0, reach=0.5}
  [968] = {accel=30, decel=30, tmax=100, leave=0, reach=0.5}
  [969] = {accel=30, decel=30, tmax=100, leave=0, reach=0.5}
  [970] = {accel=30, decel=30, tmax=100, leave=0, reach=0.5}
  [971] = {accel=30, decel=30, tmax=100, leave=0, reach=0.5}
  [972] = {accel=30, decel=30, tmax=100, leave=0, reach=0.5}
  [973] = {accel=30, decel=30, tmax=100, leave=0, reach=0.5}
  [974] = {accel=30, decel=30, tmax=100, leave=0, reach=0.5}
  [975] = {accel=30, decel=30, tmax=100, leave=0, reach=0.5}
  [976] = {accel=30, decel=30, tmax=100, leave=0, reach=0.5}
  [977] = {accel=30, decel=30, tmax=100, leave=0, reach=0.5}
  [978] = {accel=30, decel=30, tmax=100, leave=0, reach=0.5}
  [979] = {accel=30, decel=30, tmax=100, leave=0, reach=0.5}
  [980] = {accel=30, decel=30, tmax=100, leave=0, reach=0.5}
  [981] = {accel=30, decel=30, tmax=100, leave=0, reach=0.5}
  [982] = {accel=30, decel=30, tmax=100, leave=0, reach=0.5}
  [983] = {accel=30, decel=30, tmax=100, leave=0, reach=0.5}
  [984] = {accel=30, decel=30, tmax=100, leave=0, reach=0.5}
  [985] = {accel=30, decel=30, tmax=100, leave=0, reach=0.5}
  [986] = {accel=30, decel=30, tmax=100, leave=0, reach=0.5}
  [987] = {accel=30, decel=30, tmax=100, leave=0, reach=0.5}
  [988] = {accel=30, decel=30, tmax=100, leave=0, reach=0.5}
  [989] = {accel=30, decel=30, tmax=100, leave=0, reach=0.5}
  [990] = {accel=30, decel=30, tmax=100, leave=0, reach=0.5}
  [991] = {accel=30, decel=30, tmax=100, leave=0, reach=0.5}
  [992] = {accel=30, decel=30, tmax=100, leave=0, reach=0.5}
  [993] = {accel=30, decel=30, tmax=100, leave=0, reach=0.5}
  [994] = {accel=30, decel=30, tmax=100, leave=0, reach=0.5}
  [995] = {accel=30, decel=30, tmax=100, leave=0, reach=0.5}
  [996] = {accel=30, decel=30, tmax=100, leave=0, reach=0.5}
  [997] = {accel=30, decel=30, tmax=100, leave=0, reach=0.5}
  [998] = {accel=30, decel=30, tmax=100, leave=0, reach=0.5}
  [999] = {accel=30, decel=30, tmax=100, leave=0, reach=0.5}
num K = 35
num nCountCycle = 1
public num nCurrentTraj
num nCurtRadius
num nDistToOrign = 225.000310635
num nFileId
num nFileId2 = 1
num nHundredRead
num nHundredWrite
public num nMoveID
public num nPrdRadius = 50.0559565
num nPtBuffer = 500
num nPtOfTraj[16]
num nReadJnt = 1
public num nReadPtr = 1
public num nSpdOfTCP = 5.399736
public num nTabSpdCode
public num nThousandRead
public num nThousandWrite
num nTime[2]
  [0] = 1611.967
  [1] = -4198.782
public num nTotalTrajs = 1
public num nTrajofRead
num nWriteJnt = 1
public num nWritePtr = 902
public num nZshift
pointRx pGrinding = {x=-21.338, y=-123.132, z=55.455, rx=-4.904, ry=-179.25, rz=-65, fatherId=fPrdFrame[0]}
pointRx pPBuff = {fatherId=world[0]}
pointRx pPointRead[1000]
  [0] = {x=-12.659, y=-28.385, z=13.978, rx=178.274, ry=-0.79, rz=135.169, fatherId=fPrdFrame[0]}
  [1] = {x=-21.338, y=-123.132, z=55.455, rx=175.096, ry=-0.75, rz=115, fatherId=fPrdFrame[0]}
  [2] = {x=-21.338, y=-123.132, z=5.455, rx=175.096, ry=-0.75, rz=115, fatherId=fPrdFrame[0]}
  [3] = {x=-19.855, y=-123.132, z=5.437, rx=175.096, ry=-0.691, rz=115, fatherId=fPrdFrame[0]}
  [4] = {x=-18.372, y=-123.132, z=5.419, rx=175.096, ry=-0.632, rz=115, fatherId=fPrdFrame[0]}
  [5] = {x=-16.888, y=-123.132, z=5.404, rx=175.096, ry=-0.573, rz=115, fatherId=fPrdFrame[0]}
  [6] = {x=-15.405, y=-123.132, z=5.389, rx=175.096, ry=-0.513, rz=115, fatherId=fPrdFrame[0]}
  [7] = {x=-13.921, y=-123.132, z=5.377, rx=175.096, ry=-0.454, rz=115, fatherId=fPrdFrame[0]}
  [8] = {x=-12.438, y=-123.132, z=5.366, rx=175.096, ry=-0.395, rz=115, fatherId=fPrdFrame[0]}
  [9] = {x=-10.954, y=-123.132, z=5.356, rx=175.096, ry=-0.336, rz=115, fatherId=fPrdFrame[0]}
  [10] = {x=-9.471, y=-123.132, z=5.348, rx=175.096, ry=-0.277, rz=115, fatherId=fPrdFrame[0]}
  [11] = {x=-7.987, y=-123.132, z=5.341, rx=175.096, ry=-0.217, rz=115, fatherId=fPrdFrame[0]}
  [12] = {x=-6.504, y=-123.132, z=5.337, rx=175.096, ry=-0.158, rz=115, fatherId=fPrdFrame[0]}
  [13] = {x=-5.02, y=-123.132, z=5.333, rx=175.096, ry=-0.099, rz=115, fatherId=fPrdFrame[0]}
  [14] = {x=-3.537, y=-123.132, z=5.331, rx=175.096, ry=-0.04, rz=115, fatherId=fPrdFrame[0]}
  [15] = {x=-2.053, y=-123.132, z=5.331, rx=175.096, ry=0.02, rz=115, fatherId=fPrdFrame[0]}
  [16] = {x=-0.57, y=-123.132, z=5.332, rx=175.096, ry=0.079, rz=115, fatherId=fPrdFrame[0]}
  [17] = {x=0.913, y=-123.132, z=5.335, rx=175.096, ry=0.138, rz=115, fatherId=fPrdFrame[0]}
  [18] = {x=2.397, y=-123.132, z=5.34, rx=175.096, ry=0.197, rz=115, fatherId=fPrdFrame[0]}
  [19] = {x=3.88, y=-123.132, z=5.346, rx=175.096, ry=0.256, rz=115, fatherId=fPrdFrame[0]}
  [20] = {x=5.364, y=-123.132, z=5.353, rx=175.096, ry=0.316, rz=115, fatherId=fPrdFrame[0]}
  [21] = {x=6.847, y=-123.132, z=5.362, rx=175.096, ry=0.375, rz=115, fatherId=fPrdFrame[0]}
  [22] = {x=8.331, y=-123.132, z=5.373, rx=175.096, ry=0.434, rz=115, fatherId=fPrdFrame[0]}
  [23] = {x=9.814, y=-123.132, z=5.385, rx=175.096, ry=0.493, rz=115, fatherId=fPrdFrame[0]}
  [24] = {x=11.298, y=-123.132, z=5.399, rx=175.096, ry=0.553, rz=115, fatherId=fPrdFrame[0]}
  [25] = {x=12.781, y=-123.132, z=5.414, rx=175.096, ry=0.612, rz=115, fatherId=fPrdFrame[0]}
  [26] = {x=14.265, y=-123.132, z=5.431, rx=175.096, ry=0.671, rz=115, fatherId=fPrdFrame[0]}
  [27] = {x=15.748, y=-123.132, z=5.449, rx=175.096, ry=0.73, rz=115, fatherId=fPrdFrame[0]}
  [28] = {x=24.649, y=-121.649, z=5.464, rx=175.155, ry=1.086, rz=115, fatherId=fPrdFrame[0]}
  [29] = {x=23.165, y=-121.649, z=5.436, rx=175.155, ry=1.026, rz=115, fatherId=fPrdFrame[0]}
  [30] = {x=21.682, y=-121.649, z=5.41, rx=175.155, ry=0.967, rz=115, fatherId=fPrdFrame[0]}
  [31] = {x=20.198, y=-121.649, z=5.385, rx=175.155, ry=0.908, rz=115, fatherId=fPrdFrame[0]}
  [32] = {x=18.715, y=-121.649, z=5.362, rx=175.155, ry=0.849, rz=115, fatherId=fPrdFrame[0]}
  [33] = {x=17.232, y=-121.649, z=5.341, rx=175.155, ry=0.789, rz=115, fatherId=fPrdFrame[0]}
  [34] = {x=15.748, y=-121.649, z=5.321, rx=175.155, ry=0.73, rz=115, fatherId=fPrdFrame[0]}
  [35] = {x=14.265, y=-121.649, z=5.303, rx=175.155, ry=0.671, rz=115, fatherId=fPrdFrame[0]}
  [36] = {x=12.781, y=-121.649, z=5.286, rx=175.155, ry=0.612, rz=115, fatherId=fPrdFrame[0]}
  [37] = {x=11.298, y=-121.649, z=5.271, rx=175.155, ry=0.553, rz=115, fatherId=fPrdFrame[0]}
  [38] = {x=9.814, y=-121.649, z=5.257, rx=175.155, ry=0.493, rz=115, fatherId=fPrdFrame[0]}
  [39] = {x=8.331, y=-121.649, z=5.245, rx=175.155, ry=0.434, rz=115, fatherId=fPrdFrame[0]}
  [40] = {x=6.847, y=-121.649, z=5.234, rx=175.155, ry=0.375, rz=115, fatherId=fPrdFrame[0]}
  [41] = {x=5.364, y=-121.649, z=5.225, rx=175.155, ry=0.316, rz=115, fatherId=fPrdFrame[0]}
  [42] = {x=3.88, y=-121.649, z=5.218, rx=175.155, ry=0.256, rz=115, fatherId=fPrdFrame[0]}
  [43] = {x=2.397, y=-121.649, z=5.212, rx=175.155, ry=0.197, rz=115, fatherId=fPrdFrame[0]}
  [44] = {x=0.913, y=-121.649, z=5.207, rx=175.155, ry=0.138, rz=115, fatherId=fPrdFrame[0]}
  [45] = {x=-0.57, y=-121.649, z=5.204, rx=175.155, ry=0.079, rz=115, fatherId=fPrdFrame[0]}
  [46] = {x=-2.053, y=-121.649, z=5.203, rx=175.155, ry=0.02, rz=115, fatherId=fPrdFrame[0]}
  [47] = {x=-3.537, y=-121.649, z=5.203, rx=175.155, ry=-0.04, rz=115, fatherId=fPrdFrame[0]}
  [48] = {x=-5.02, y=-121.649, z=5.205, rx=175.155, ry=-0.099, rz=115, fatherId=fPrdFrame[0]}
  [49] = {x=-6.504, y=-121.649, z=5.209, rx=175.155, ry=-0.158, rz=115, fatherId=fPrdFrame[0]}
  [50] = {x=-7.987, y=-121.649, z=5.214, rx=175.155, ry=-0.217, rz=115, fatherId=fPrdFrame[0]}
  [51] = {x=-9.471, y=-121.649, z=5.22, rx=175.155, ry=-0.277, rz=115, fatherId=fPrdFrame[0]}
  [52] = {x=-10.954, y=-121.649, z=5.228, rx=175.155, ry=-0.336, rz=115, fatherId=fPrdFrame[0]}
  [53] = {x=-12.438, y=-121.649, z=5.238, rx=175.155, ry=-0.395, rz=115, fatherId=fPrdFrame[0]}
  [54] = {x=-13.921, y=-121.649, z=5.249, rx=175.155, ry=-0.454, rz=115, fatherId=fPrdFrame[0]}
  [55] = {x=-15.405, y=-121.649, z=5.261, rx=175.155, ry=-0.513, rz=115, fatherId=fPrdFrame[0]}
  [56] = {x=-16.888, y=-121.649, z=5.276, rx=175.155, ry=-0.573, rz=115, fatherId=fPrdFrame[0]}
  [57] = {x=-18.372, y=-121.649, z=5.291, rx=175.155, ry=-0.632, rz=115, fatherId=fPrdFrame[0]}
  [58] = {x=-19.855, y=-121.649, z=5.309, rx=175.155, ry=-0.691, rz=115, fatherId=fPrdFrame[0]}
  [59] = {x=-21.338, y=-121.649, z=5.328, rx=175.155, ry=-0.75, rz=115, fatherId=fPrdFrame[0]}
  [60] = {x=-22.822, y=-121.649, z=5.348, rx=175.155, ry=-0.81, rz=115, fatherId=fPrdFrame[0]}
  [61] = {x=-24.305, y=-121.649, z=5.37, rx=175.155, ry=-0.869, rz=115, fatherId=fPrdFrame[0]}
  [62] = {x=-25.789, y=-121.649, z=5.393, rx=175.155, ry=-0.928, rz=115, fatherId=fPrdFrame[0]}
  [63] = {x=-27.272, y=-121.649, z=5.419, rx=175.155, ry=-0.987, rz=115, fatherId=fPrdFrame[0]}
  [64] = {x=-28.756, y=-121.649, z=5.445, rx=175.155, ry=-1.046, rz=115, fatherId=fPrdFrame[0]}
  [65] = {x=-36.173, y=-120.165, z=5.475, rx=175.213, ry=-1.343, rz=115, fatherId=fPrdFrame[0]}
  [66] = {x=-34.69, y=-120.165, z=5.441, rx=175.213, ry=-1.283, rz=115, fatherId=fPrdFrame[0]}
  [67] = {x=-33.206, y=-120.165, z=5.408, rx=175.214, ry=-1.224, rz=115, fatherId=fPrdFrame[0]}
  [68] = {x=-31.723, y=-120.165, z=5.377, rx=175.214, ry=-1.165, rz=115, fatherId=fPrdFrame[0]}
  [69] = {x=-30.239, y=-120.165, z=5.347, rx=175.214, ry=-1.106, rz=115, fatherId=fPrdFrame[0]}
  [70] = {x=-28.756, y=-120.165, z=5.319, rx=175.214, ry=-1.046, rz=115, fatherId=fPrdFrame[0]}
  [71] = {x=-27.272, y=-120.165, z=5.292, rx=175.214, ry=-0.987, rz=115, fatherId=fPrdFrame[0]}
  [72] = {x=-25.789, y=-120.165, z=5.267, rx=175.214, ry=-0.928, rz=115, fatherId=fPrdFrame[0]}
  [73] = {x=-24.305, y=-120.165, z=5.244, rx=175.214, ry=-0.869, rz=115, fatherId=fPrdFrame[0]}
  [74] = {x=-22.822, y=-120.165, z=5.222, rx=175.214, ry=-0.81, rz=115, fatherId=fPrdFrame[0]}
  [75] = {x=-21.338, y=-120.165, z=5.201, rx=175.214, ry=-0.75, rz=115, fatherId=fPrdFrame[0]}
  [76] = {x=-19.855, y=-120.165, z=5.182, rx=175.214, ry=-0.691, rz=115, fatherId=fPrdFrame[0]}
  [77] = {x=-18.372, y=-120.165, z=5.165, rx=175.214, ry=-0.632, rz=115, fatherId=fPrdFrame[0]}
  [78] = {x=-16.888, y=-120.165, z=5.149, rx=175.214, ry=-0.573, rz=115, fatherId=fPrdFrame[0]}
  [79] = {x=-15.405, y=-120.165, z=5.135, rx=175.214, ry=-0.513, rz=115, fatherId=fPrdFrame[0]}
  [80] = {x=-13.921, y=-120.165, z=5.122, rx=175.215, ry=-0.454, rz=115, fatherId=fPrdFrame[0]}
  [81] = {x=-12.438, y=-120.165, z=5.111, rx=175.215, ry=-0.395, rz=115, fatherId=fPrdFrame[0]}
  [82] = {x=-10.954, y=-120.165, z=5.102, rx=175.215, ry=-0.336, rz=115, fatherId=fPrdFrame[0]}
  [83] = {x=-9.471, y=-120.165, z=5.094, rx=175.215, ry=-0.277, rz=115, fatherId=fPrdFrame[0]}
  [84] = {x=-7.987, y=-120.165, z=5.087, rx=175.215, ry=-0.217, rz=115, fatherId=fPrdFrame[0]}
  [85] = {x=-6.504, y=-120.165, z=5.082, rx=175.215, ry=-0.158, rz=115, fatherId=fPrdFrame[0]}
  [86] = {x=-5.02, y=-120.165, z=5.079, rx=175.215, ry=-0.099, rz=115, fatherId=fPrdFrame[0]}
  [87] = {x=-3.537, y=-120.165, z=5.077, rx=175.215, ry=-0.04, rz=115, fatherId=fPrdFrame[0]}
  [88] = {x=-2.053, y=-120.165, z=5.077, rx=175.215, ry=0.02, rz=115, fatherId=fPrdFrame[0]}
  [89] = {x=-0.57, y=-120.165, z=5.078, rx=175.215, ry=0.079, rz=115, fatherId=fPrdFrame[0]}
  [90] = {x=0.913, y=-120.165, z=5.081, rx=175.215, ry=0.138, rz=115, fatherId=fPrdFrame[0]}
  [91] = {x=2.397, y=-120.165, z=5.085, rx=175.215, ry=0.197, rz=115, fatherId=fPrdFrame[0]}
  [92] = {x=3.88, y=-120.165, z=5.091, rx=175.215, ry=0.256, rz=115, fatherId=fPrdFrame[0]}
  [93] = {x=5.364, y=-120.165, z=5.099, rx=175.215, ry=0.316, rz=115, fatherId=fPrdFrame[0]}
  [94] = {x=6.847, y=-120.165, z=5.108, rx=175.215, ry=0.375, rz=115, fatherId=fPrdFrame[0]}
  [95] = {x=8.331, y=-120.165, z=5.118, rx=175.215, ry=0.434, rz=115, fatherId=fPrdFrame[0]}
  [96] = {x=9.814, y=-120.165, z=5.131, rx=175.214, ry=0.493, rz=115, fatherId=fPrdFrame[0]}
  [97] = {x=11.298, y=-120.165, z=5.144, rx=175.214, ry=0.552, rz=115, fatherId=fPrdFrame[0]}
  [98] = {x=12.781, y=-120.165, z=5.159, rx=175.214, ry=0.612, rz=115, fatherId=fPrdFrame[0]}
  [99] = {x=14.265, y=-120.165, z=5.176, rx=175.214, ry=0.671, rz=115, fatherId=fPrdFrame[0]}
  [100] = {x=15.748, y=-120.165, z=5.195, rx=175.214, ry=0.73, rz=115, fatherId=fPrdFrame[0]}
  [101] = {x=17.232, y=-120.165, z=5.215, rx=175.214, ry=0.789, rz=115, fatherId=fPrdFrame[0]}
  [102] = {x=18.715, y=-120.165, z=5.236, rx=175.214, ry=0.849, rz=115, fatherId=fPrdFrame[0]}
  [103] = {x=20.199, y=-120.165, z=5.259, rx=175.214, ry=0.908, rz=115, fatherId=fPrdFrame[0]}
  [104] = {x=21.682, y=-120.165, z=5.283, rx=175.214, ry=0.967, rz=115, fatherId=fPrdFrame[0]}
  [105] = {x=23.165, y=-120.165, z=5.31, rx=175.214, ry=1.026, rz=115, fatherId=fPrdFrame[0]}
  [106] = {x=24.649, y=-120.165, z=5.337, rx=175.214, ry=1.085, rz=115, fatherId=fPrdFrame[0]}
  [107] = {x=26.132, y=-120.165, z=5.366, rx=175.214, ry=1.145, rz=115, fatherId=fPrdFrame[0]}
  [108] = {x=27.616, y=-120.165, z=5.397, rx=175.214, ry=1.204, rz=115, fatherId=fPrdFrame[0]}
  [109] = {x=29.099, y=-120.165, z=5.429, rx=175.214, ry=1.263, rz=115, fatherId=fPrdFrame[0]}
  [110] = {x=30.583, y=-120.165, z=5.463, rx=175.213, ry=1.322, rz=115, fatherId=fPrdFrame[0]}
  [111] = {x=35.033, y=-118.681, z=5.449, rx=175.272, ry=1.5, rz=115, fatherId=fPrdFrame[0]}
  [112] = {x=33.55, y=-118.681, z=5.411, rx=175.272, ry=1.441, rz=115, fatherId=fPrdFrame[0]}
  [113] = {x=32.066, y=-118.681, z=5.374, rx=175.273, ry=1.382, rz=115, fatherId=fPrdFrame[0]}
  [114] = {x=30.583, y=-118.681, z=5.339, rx=175.273, ry=1.322, rz=115, fatherId=fPrdFrame[0]}
  [115] = {x=29.099, y=-118.681, z=5.305, rx=175.273, ry=1.263, rz=115, fatherId=fPrdFrame[0]}
  [116] = {x=27.616, y=-118.681, z=5.272, rx=175.273, ry=1.204, rz=115, fatherId=fPrdFrame[0]}
  [117] = {x=26.132, y=-118.681, z=5.242, rx=175.273, ry=1.145, rz=115, fatherId=fPrdFrame[0]}
  [118] = {x=24.649, y=-118.681, z=5.212, rx=175.273, ry=1.085, rz=115, fatherId=fPrdFrame[0]}
  [119] = {x=23.165, y=-118.682, z=5.185, rx=175.273, ry=1.026, rz=115, fatherId=fPrdFrame[0]}
  [120] = {x=21.682, y=-118.682, z=5.159, rx=175.273, ry=0.967, rz=115, fatherId=fPrdFrame[0]}
  [121] = {x=20.199, y=-118.682, z=5.134, rx=175.273, ry=0.908, rz=115, fatherId=fPrdFrame[0]}
  [122] = {x=18.715, y=-118.682, z=5.111, rx=175.273, ry=0.849, rz=115, fatherId=fPrdFrame[0]}
  [123] = {x=17.232, y=-118.682, z=5.09, rx=175.273, ry=0.789, rz=115, fatherId=fPrdFrame[0]}
  [124] = {x=15.748, y=-118.682, z=5.07, rx=175.274, ry=0.73, rz=115, fatherId=fPrdFrame[0]}
  [125] = {x=14.265, y=-118.682, z=5.051, rx=175.274, ry=0.671, rz=115, fatherId=fPrdFrame[0]}
  [126] = {x=12.781, y=-118.682, z=5.035, rx=175.274, ry=0.612, rz=115, fatherId=fPrdFrame[0]}
  [127] = {x=11.298, y=-118.682, z=5.019, rx=175.274, ry=0.552, rz=115, fatherId=fPrdFrame[0]}
  [128] = {x=9.814, y=-118.682, z=5.006, rx=175.274, ry=0.493, rz=115, fatherId=fPrdFrame[0]}
  [129] = {x=8.331, y=-118.682, z=4.994, rx=175.274, ry=0.434, rz=115, fatherId=fPrdFrame[0]}
  [130] = {x=6.847, y=-118.682, z=4.983, rx=175.274, ry=0.375, rz=115, fatherId=fPrdFrame[0]}
  [131] = {x=5.364, y=-118.682, z=4.974, rx=175.274, ry=0.316, rz=115, fatherId=fPrdFrame[0]}
  [132] = {x=3.88, y=-118.682, z=4.967, rx=175.274, ry=0.256, rz=115, fatherId=fPrdFrame[0]}
  [133] = {x=2.397, y=-118.682, z=4.961, rx=175.274, ry=0.197, rz=115, fatherId=fPrdFrame[0]}
  [134] = {x=0.913, y=-118.682, z=4.956, rx=175.274, ry=0.138, rz=115, fatherId=fPrdFrame[0]}
  [135] = {x=-0.57, y=-118.682, z=4.953, rx=175.274, ry=0.079, rz=115, fatherId=fPrdFrame[0]}
  [136] = {x=-2.053, y=-118.682, z=4.952, rx=175.274, ry=0.02, rz=115, fatherId=fPrdFrame[0]}
  [137] = {x=-3.537, y=-118.682, z=4.952, rx=175.274, ry=-0.04, rz=115, fatherId=fPrdFrame[0]}
  [138] = {x=-5.02, y=-118.682, z=4.954, rx=175.274, ry=-0.099, rz=115, fatherId=fPrdFrame[0]}
  [139] = {x=-6.504, y=-118.682, z=4.958, rx=175.274, ry=-0.158, rz=115, fatherId=fPrdFrame[0]}
  [140] = {x=-7.987, y=-118.682, z=4.962, rx=175.274, ry=-0.217, rz=115, fatherId=fPrdFrame[0]}
  [141] = {x=-9.471, y=-118.682, z=4.969, rx=175.274, ry=-0.277, rz=115, fatherId=fPrdFrame[0]}
  [142] = {x=-10.954, y=-118.682, z=4.977, rx=175.274, ry=-0.336, rz=115, fatherId=fPrdFrame[0]}
  [143] = {x=-12.438, y=-118.682, z=4.986, rx=175.274, ry=-0.395, rz=115, fatherId=fPrdFrame[0]}
  [144] = {x=-13.921, y=-118.682, z=4.998, rx=175.274, ry=-0.454, rz=115, fatherId=fPrdFrame[0]}
  [145] = {x=-15.405, y=-118.682, z=5.01, rx=175.274, ry=-0.513, rz=115, fatherId=fPrdFrame[0]}
  [146] = {x=-16.888, y=-118.682, z=5.024, rx=175.274, ry=-0.573, rz=115, fatherId=fPrdFrame[0]}
  [147] = {x=-18.372, y=-118.682, z=5.04, rx=175.274, ry=-0.632, rz=115, fatherId=fPrdFrame[0]}
  [148] = {x=-19.855, y=-118.682, z=5.058, rx=175.274, ry=-0.691, rz=115, fatherId=fPrdFrame[0]}
  [149] = {x=-21.339, y=-118.682, z=5.076, rx=175.273, ry=-0.75, rz=115, fatherId=fPrdFrame[0]}
  [150] = {x=-22.822, y=-118.682, z=5.097, rx=175.273, ry=-0.809, rz=115, fatherId=fPrdFrame[0]}
  [151] = {x=-24.305, y=-118.682, z=5.119, rx=175.273, ry=-0.869, rz=115, fatherId=fPrdFrame[0]}
  [152] = {x=-25.789, y=-118.682, z=5.142, rx=175.273, ry=-0.928, rz=115, fatherId=fPrdFrame[0]}
  [153] = {x=-27.272, y=-118.682, z=5.167, rx=175.273, ry=-0.987, rz=115, fatherId=fPrdFrame[0]}
  [154] = {x=-28.756, y=-118.681, z=5.194, rx=175.273, ry=-1.046, rz=115, fatherId=fPrdFrame[0]}
  [155] = {x=-30.239, y=-118.681, z=5.222, rx=175.273, ry=-1.106, rz=115, fatherId=fPrdFrame[0]}
  [156] = {x=-31.723, y=-118.681, z=5.252, rx=175.273, ry=-1.165, rz=115, fatherId=fPrdFrame[0]}
  [157] = {x=-33.206, y=-118.681, z=5.283, rx=175.273, ry=-1.224, rz=115, fatherId=fPrdFrame[0]}
  [158] = {x=-34.69, y=-118.681, z=5.316, rx=175.273, ry=-1.283, rz=115, fatherId=fPrdFrame[0]}
  [159] = {x=-36.173, y=-118.681, z=5.35, rx=175.273, ry=-1.342, rz=115, fatherId=fPrdFrame[0]}
  [160] = {x=-37.657, y=-118.681, z=5.386, rx=175.272, ry=-1.402, rz=115, fatherId=fPrdFrame[0]}
  [161] = {x=-39.14, y=-118.681, z=5.424, rx=175.272, ry=-1.461, rz=115, fatherId=fPrdFrame[0]}
  [162] = {x=-40.624, y=-118.681, z=5.463, rx=175.272, ry=-1.52, rz=115, fatherId=fPrdFrame[0]}
  [163] = {x=-45.074, y=-117.198, z=5.466, rx=175.331, ry=-1.698, rz=115, fatherId=fPrdFrame[0]}
  [164] = {x=-43.591, y=-117.198, z=5.422, rx=175.331, ry=-1.638, rz=115, fatherId=fPrdFrame[0]}
  [165] = {x=-42.107, y=-117.198, z=5.38, rx=175.331, ry=-1.579, rz=115, fatherId=fPrdFrame[0]}
  [166] = {x=-40.624, y=-117.198, z=5.34, rx=175.331, ry=-1.52, rz=115, fatherId=fPrdFrame[0]}
  [167] = {x=-39.14, y=-117.198, z=5.3, rx=175.332, ry=-1.461, rz=115, fatherId=fPrdFrame[0]}
  [168] = {x=-37.657, y=-117.198, z=5.263, rx=175.332, ry=-1.402, rz=115, fatherId=fPrdFrame[0]}
  [169] = {x=-36.173, y=-117.198, z=5.227, rx=175.332, ry=-1.342, rz=115, fatherId=fPrdFrame[0]}
  [170] = {x=-34.69, y=-117.198, z=5.193, rx=175.332, ry=-1.283, rz=115, fatherId=fPrdFrame[0]}
  [171] = {x=-33.206, y=-117.198, z=5.16, rx=175.332, ry=-1.224, rz=115, fatherId=fPrdFrame[0]}
  [172] = {x=-31.723, y=-117.198, z=5.129, rx=175.332, ry=-1.165, rz=115, fatherId=fPrdFrame[0]}
  [173] = {x=-30.239, y=-117.198, z=5.099, rx=175.332, ry=-1.105, rz=115, fatherId=fPrdFrame[0]}
  [174] = {x=-28.756, y=-117.198, z=5.071, rx=175.332, ry=-1.046, rz=115, fatherId=fPrdFrame[0]}
  [175] = {x=-27.272, y=-117.198, z=5.044, rx=175.332, ry=-0.987, rz=115, fatherId=fPrdFrame[0]}
  [176] = {x=-25.789, y=-117.198, z=5.019, rx=175.332, ry=-0.928, rz=115, fatherId=fPrdFrame[0]}
  [177] = {x=-24.305, y=-117.198, z=4.996, rx=175.333, ry=-0.869, rz=115, fatherId=fPrdFrame[0]}
  [178] = {x=-22.822, y=-117.198, z=4.974, rx=175.333, ry=-0.809, rz=115, fatherId=fPrdFrame[0]}
  [179] = {x=-21.339, y=-117.198, z=4.953, rx=175.333, ry=-0.75, rz=115, fatherId=fPrdFrame[0]}
  [180] = {x=-19.855, y=-117.198, z=4.934, rx=175.333, ry=-0.691, rz=115, fatherId=fPrdFrame[0]}
  [181] = {x=-18.372, y=-117.198, z=4.917, rx=175.333, ry=-0.632, rz=115, fatherId=fPrdFrame[0]}
  [182] = {x=-16.888, y=-117.198, z=4.901, rx=175.333, ry=-0.573, rz=115, fatherId=fPrdFrame[0]}
  [183] = {x=-15.405, y=-117.198, z=4.887, rx=175.333, ry=-0.513, rz=115, fatherId=fPrdFrame[0]}
  [184] = {x=-13.921, y=-117.198, z=4.874, rx=175.333, ry=-0.454, rz=115, fatherId=fPrdFrame[0]}
  [185] = {x=-12.438, y=-117.198, z=4.863, rx=175.333, ry=-0.395, rz=115, fatherId=fPrdFrame[0]}
  [186] = {x=-10.954, y=-117.198, z=4.854, rx=175.333, ry=-0.336, rz=115, fatherId=fPrdFrame[0]}
  [187] = {x=-9.471, y=-117.198, z=4.846, rx=175.333, ry=-0.276, rz=115, fatherId=fPrdFrame[0]}
  [188] = {x=-7.987, y=-117.198, z=4.839, rx=175.333, ry=-0.217, rz=115, fatherId=fPrdFrame[0]}
  [189] = {x=-6.504, y=-117.198, z=4.834, rx=175.333, ry=-0.158, rz=115, fatherId=fPrdFrame[0]}
  [190] = {x=-5.02, y=-117.198, z=4.831, rx=175.333, ry=-0.099, rz=115, fatherId=fPrdFrame[0]}
  [191] = {x=-3.537, y=-117.198, z=4.829, rx=175.333, ry=-0.04, rz=115, fatherId=fPrdFrame[0]}
  [192] = {x=-2.053, y=-117.198, z=4.829, rx=175.333, ry=0.02, rz=115, fatherId=fPrdFrame[0]}
  [193] = {x=-0.57, y=-117.198, z=4.83, rx=175.333, ry=0.079, rz=115, fatherId=fPrdFrame[0]}
  [194] = {x=0.913, y=-117.198, z=4.833, rx=175.333, ry=0.138, rz=115, fatherId=fPrdFrame[0]}
  [195] = {x=2.397, y=-117.198, z=4.837, rx=175.333, ry=0.197, rz=115, fatherId=fPrdFrame[0]}
  [196] = {x=3.88, y=-117.198, z=4.843, rx=175.333, ry=0.256, rz=115, fatherId=fPrdFrame[0]}
  [197] = {x=5.364, y=-117.198, z=4.851, rx=175.333, ry=0.316, rz=115, fatherId=fPrdFrame[0]}
  [198] = {x=6.847, y=-117.198, z=4.86, rx=175.333, ry=0.375, rz=115, fatherId=fPrdFrame[0]}
  [199] = {x=8.331, y=-117.198, z=4.87, rx=175.333, ry=0.434, rz=115, fatherId=fPrdFrame[0]}
  [200] = {x=9.814, y=-117.198, z=4.883, rx=175.333, ry=0.493, rz=115, fatherId=fPrdFrame[0]}
  [201] = {x=11.298, y=-117.198, z=4.896, rx=175.333, ry=0.552, rz=115, fatherId=fPrdFrame[0]}
  [202] = {x=12.781, y=-117.198, z=4.911, rx=175.333, ry=0.612, rz=115, fatherId=fPrdFrame[0]}
  [203] = {x=14.265, y=-117.198, z=4.928, rx=175.333, ry=0.671, rz=115, fatherId=fPrdFrame[0]}
  [204] = {x=15.748, y=-117.198, z=4.947, rx=175.333, ry=0.73, rz=115, fatherId=fPrdFrame[0]}
  [205] = {x=17.232, y=-117.198, z=4.966, rx=175.333, ry=0.789, rz=115, fatherId=fPrdFrame[0]}
  [206] = {x=18.715, y=-117.198, z=4.988, rx=175.333, ry=0.848, rz=115, fatherId=fPrdFrame[0]}
  [207] = {x=20.199, y=-117.198, z=5.011, rx=175.333, ry=0.908, rz=115, fatherId=fPrdFrame[0]}
  [208] = {x=21.682, y=-117.198, z=5.035, rx=175.332, ry=0.967, rz=115, fatherId=fPrdFrame[0]}
  [209] = {x=23.165, y=-117.198, z=5.062, rx=175.332, ry=1.026, rz=115, fatherId=fPrdFrame[0]}
  [210] = {x=24.649, y=-117.198, z=5.089, rx=175.332, ry=1.085, rz=115, fatherId=fPrdFrame[0]}
  [211] = {x=26.132, y=-117.198, z=5.118, rx=175.332, ry=1.145, rz=115, fatherId=fPrdFrame[0]}
  [212] = {x=27.616, y=-117.198, z=5.149, rx=175.332, ry=1.204, rz=115, fatherId=fPrdFrame[0]}
  [213] = {x=29.099, y=-117.198, z=5.181, rx=175.332, ry=1.263, rz=115, fatherId=fPrdFrame[0]}
  [214] = {x=30.583, y=-117.198, z=5.215, rx=175.332, ry=1.322, rz=115, fatherId=fPrdFrame[0]}
  [215] = {x=32.066, y=-117.198, z=5.251, rx=175.332, ry=1.381, rz=115, fatherId=fPrdFrame[0]}
  [216] = {x=33.55, y=-117.198, z=5.288, rx=175.332, ry=1.441, rz=115, fatherId=fPrdFrame[0]}
  [217] = {x=35.033, y=-117.198, z=5.326, rx=175.332, ry=1.5, rz=115, fatherId=fPrdFrame[0]}
  [218] = {x=36.517, y=-117.198, z=5.366, rx=175.331, ry=1.559, rz=115, fatherId=fPrdFrame[0]}
  [219] = {x=38, y=-117.198, z=5.408, rx=175.331, ry=1.618, rz=115, fatherId=fPrdFrame[0]}
  [220] = {x=39.484, y=-117.198, z=5.451, rx=175.331, ry=1.678, rz=115, fatherId=fPrdFrame[0]}
  [221] = {x=43.934, y=-115.714, z=5.468, rx=175.39, ry=1.855, rz=115, fatherId=fPrdFrame[0]}
  [222] = {x=42.451, y=-115.714, z=5.42, rx=175.39, ry=1.796, rz=115, fatherId=fPrdFrame[0]}
  [223] = {x=40.967, y=-115.714, z=5.374, rx=175.39, ry=1.737, rz=115, fatherId=fPrdFrame[0]}
  [224] = {x=39.484, y=-115.714, z=5.329, rx=175.39, ry=1.677, rz=115, fatherId=fPrdFrame[0]}
  [225] = {x=38, y=-115.714, z=5.286, rx=175.39, ry=1.618, rz=115, fatherId=fPrdFrame[0]}
  [226] = {x=36.517, y=-115.714, z=5.244, rx=175.391, ry=1.559, rz=115, fatherId=fPrdFrame[0]}
  [227] = {x=35.033, y=-115.714, z=5.204, rx=175.391, ry=1.5, rz=115, fatherId=fPrdFrame[0]}
  [228] = {x=33.55, y=-115.714, z=5.166, rx=175.391, ry=1.441, rz=115, fatherId=fPrdFrame[0]}
  [229] = {x=32.066, y=-115.714, z=5.129, rx=175.391, ry=1.381, rz=115, fatherId=fPrdFrame[0]}
  [230] = {x=30.583, y=-115.714, z=5.094, rx=175.391, ry=1.322, rz=115, fatherId=fPrdFrame[0]}
  [231] = {x=29.099, y=-115.714, z=5.06, rx=175.391, ry=1.263, rz=115, fatherId=fPrdFrame[0]}
  [232] = {x=27.616, y=-115.714, z=5.027, rx=175.391, ry=1.204, rz=115, fatherId=fPrdFrame[0]}
  [233] = {x=26.132, y=-115.714, z=4.997, rx=175.391, ry=1.144, rz=115, fatherId=fPrdFrame[0]}
  [234] = {x=24.649, y=-115.714, z=4.967, rx=175.391, ry=1.085, rz=115, fatherId=fPrdFrame[0]}
  [235] = {x=23.166, y=-115.714, z=4.94, rx=175.392, ry=1.026, rz=115, fatherId=fPrdFrame[0]}
  [236] = {x=21.682, y=-115.714, z=4.914, rx=175.392, ry=0.967, rz=115, fatherId=fPrdFrame[0]}
  [237] = {x=20.199, y=-115.715, z=4.889, rx=175.392, ry=0.908, rz=115, fatherId=fPrdFrame[0]}
  [238] = {x=18.715, y=-115.715, z=4.866, rx=175.392, ry=0.848, rz=115, fatherId=fPrdFrame[0]}
  [239] = {x=17.232, y=-115.715, z=4.845, rx=175.392, ry=0.789, rz=115, fatherId=fPrdFrame[0]}
  [240] = {x=15.748, y=-115.715, z=4.825, rx=175.392, ry=0.73, rz=115, fatherId=fPrdFrame[0]}
  [241] = {x=14.265, y=-115.715, z=4.807, rx=175.392, ry=0.671, rz=115, fatherId=fPrdFrame[0]}
  [242] = {x=12.781, y=-115.715, z=4.79, rx=175.392, ry=0.612, rz=115, fatherId=fPrdFrame[0]}
  [243] = {x=11.298, y=-115.715, z=4.775, rx=175.392, ry=0.552, rz=115, fatherId=fPrdFrame[0]}
  [244] = {x=9.814, y=-115.715, z=4.761, rx=175.392, ry=0.493, rz=115, fatherId=fPrdFrame[0]}
  [245] = {x=8.331, y=-115.715, z=4.749, rx=175.392, ry=0.434, rz=115, fatherId=fPrdFrame[0]}
  [246] = {x=6.847, y=-115.715, z=4.738, rx=175.392, ry=0.375, rz=115, fatherId=fPrdFrame[0]}
  [247] = {x=5.364, y=-115.715, z=4.729, rx=175.392, ry=0.316, rz=115, fatherId=fPrdFrame[0]}
  [248] = {x=3.88, y=-115.715, z=4.722, rx=175.392, ry=0.256, rz=115, fatherId=fPrdFrame[0]}
  [249] = {x=2.397, y=-115.715, z=4.716, rx=175.392, ry=0.197, rz=115, fatherId=fPrdFrame[0]}
  [250] = {x=0.913, y=-115.715, z=4.711, rx=175.392, ry=0.138, rz=115, fatherId=fPrdFrame[0]}
  [251] = {x=-0.57, y=-115.715, z=4.708, rx=175.392, ry=0.079, rz=115, fatherId=fPrdFrame[0]}
  [252] = {x=-2.053, y=-115.715, z=4.707, rx=175.392, ry=0.02, rz=115, fatherId=fPrdFrame[0]}
  [253] = {x=-3.537, y=-115.715, z=4.707, rx=175.392, ry=-0.04, rz=115, fatherId=fPrdFrame[0]}
  [254] = {x=-5.02, y=-115.715, z=4.709, rx=175.392, ry=-0.099, rz=115, fatherId=fPrdFrame[0]}
  [255] = {x=-6.504, y=-115.715, z=4.713, rx=175.392, ry=-0.158, rz=115, fatherId=fPrdFrame[0]}
  [256] = {x=-7.987, y=-115.715, z=4.718, rx=175.392, ry=-0.217, rz=115, fatherId=fPrdFrame[0]}
  [257] = {x=-9.471, y=-115.715, z=4.724, rx=175.392, ry=-0.276, rz=115, fatherId=fPrdFrame[0]}
  [258] = {x=-10.954, y=-115.715, z=4.732, rx=175.392, ry=-0.336, rz=115, fatherId=fPrdFrame[0]}
  [259] = {x=-12.438, y=-115.715, z=4.742, rx=175.392, ry=-0.395, rz=115, fatherId=fPrdFrame[0]}
  [260] = {x=-13.921, y=-115.715, z=4.753, rx=175.392, ry=-0.454, rz=115, fatherId=fPrdFrame[0]}
  [261] = {x=-15.405, y=-115.715, z=4.765, rx=175.392, ry=-0.513, rz=115, fatherId=fPrdFrame[0]}
  [262] = {x=-16.888, y=-115.715, z=4.78, rx=175.392, ry=-0.572, rz=115, fatherId=fPrdFrame[0]}
  [263] = {x=-18.372, y=-115.715, z=4.795, rx=175.392, ry=-0.632, rz=115, fatherId=fPrdFrame[0]}
  [264] = {x=-19.855, y=-115.715, z=4.813, rx=175.392, ry=-0.691, rz=115, fatherId=fPrdFrame[0]}
  [265] = {x=-21.339, y=-115.715, z=4.831, rx=175.392, ry=-0.75, rz=115, fatherId=fPrdFrame[0]}
  [266] = {x=-22.822, y=-115.715, z=4.852, rx=175.392, ry=-0.809, rz=115, fatherId=fPrdFrame[0]}
  [267] = {x=-24.305, y=-115.715, z=4.874, rx=175.392, ry=-0.869, rz=115, fatherId=fPrdFrame[0]}
  [268] = {x=-25.789, y=-115.715, z=4.897, rx=175.392, ry=-0.928, rz=115, fatherId=fPrdFrame[0]}
  [269] = {x=-27.272, y=-115.714, z=4.922, rx=175.392, ry=-0.987, rz=115, fatherId=fPrdFrame[0]}
  [270] = {x=-28.756, y=-115.714, z=4.949, rx=175.392, ry=-1.046, rz=115, fatherId=fPrdFrame[0]}
  [271] = {x=-30.239, y=-115.714, z=4.977, rx=175.391, ry=-1.105, rz=115, fatherId=fPrdFrame[0]}
  [272] = {x=-31.723, y=-115.714, z=5.007, rx=175.391, ry=-1.165, rz=115, fatherId=fPrdFrame[0]}
